Universal Robots URScript: Main Program Right.script

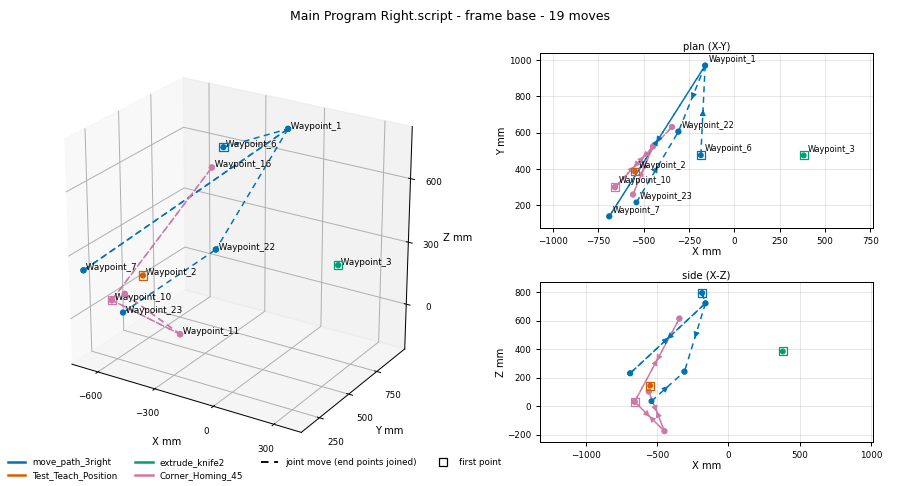
[picture p0: tool path of Main Program Right.script in frame base, 19 of 66 moves have a stored position in this frame; points joined in program order, loops and branches not executed]
def Main_Program_Right():
  global _hidden_verificationVariable=0
  set_tcp(p[0.00157,-0.09008,0.25767,0.0,0.0,0.0])
  set_safety_mode_transition_hardness(1)
  set_tool_communication(False, 115200, 0, 1, 1.5, 3.5)
  set_tool_output_mode(0)
  set_tool_digital_output_mode(0, 1)
  set_tool_digital_output_mode(1, 1)
  set_tool_voltage(0)
  set_target_payload(8.250000, [-0.001000, -0.057000, 0.067000], [0.051851, 0.051851, 0.051851, 0.000000, 0.000000, 0.000000])
  set_standard_analog_input_domain(0, 1)
  set_standard_analog_input_domain(1, 1)
  set_tool_analog_input_domain(0, 1)
  set_tool_analog_input_domain(1, 1)
  set_analog_outputdomain(0, 0)
  set_analog_outputdomain(1, 0)
  set_input_actions_to_default()
  set_gravity([0.0, 0.0, 9.82])
  global Point_1=p[0.0,0.0,0.0,0.0,0.0,0.0]
  # begin: URCap Installation Node
  #   Source: MachineLogic for Universal Robots, 3.1.7, Vention Inc.
  #   Type: MachineLogic for Universal Robots
  def waitForResponse(expected_response_vention, cname_vention):
  response_vention = socket_read_string(cname_vention,timeout=15)
  while response_vention != expected_response_vention:
  sleep(0.01)
  response_vention = socket_read_string(cname_vention,timeout=15)
  end
  sleep(0.01)
  sync()
  end
  def sendString(string_vention, expected_response_vention, cname_vention):
  socket_send_string(str_cat(string_vention,";"), cname_vention)
  response_vention = socket_read_string(cname_vention,timeout=15)
  if(response_vention == "nAck"):
  popup("nAck received")
  end
  while response_vention != expected_response_vention:
  sleep(0.01)
  response_vention = socket_read_string(cname_vention,timeout=15)
  if(response_vention == "nAck"):
  popup("nAck received")
  end
  end
  sleep(0.01)
  sync()
  end
  def sendStringNAck(string_vention, expected_response_vention, cname_vention):
  socket_send_string(str_cat(string_vention,";"), cname_vention)
  response_vention = socket_read_string(cname_vention,timeout=15)
  if(response_vention == "nAck"):
  popup("nAck received")
  end
  while(response_vention != expected_response_vention and response_vention != "nAck"):
  sleep(0.01)
  response_vention = socket_read_string(cname_vention,timeout=15)
  if(response_vention == "nAck"):
  popup("nAck received",blocking=True)
  end
  end
  sleep(0.01)
  sync()
  end
  def sendStringWithTimeout(string_vention, expected_response_vention, cname_vention):
  socket_send_string(str_cat(string_vention,";"), cname_vention)
  response_vention = socket_read_string(cname_vention,timeout=10)
  if(response_vention == "nAck"):
  popup("nAck received"+string_vention)
  end
  sleep(0.01)
  sync()
  end
  def pollString(string_vention, expected_response_vention, cname_vention):
  socket_send_string(str_cat(string_vention,";"), cname_vention)
  response_vention = socket_read_string(cname_vention,timeout=15)
  if(response_vention == "nAck"):
  popup("nAck received")
  end
  while response_vention != expected_response_vention:
  sleep(1)
  socket_send_string(str_cat(string_vention,";"), cname_vention)
  response_vention = socket_read_string(cname_vention,timeout=15)
  if(response_vention == "nAck"):
  popup("nAck received")
  end
  end
  sleep(0.01)
  sync()
  end
  def sendVariable(var_vention, data_vention, expected_response_vention, cname_vention):
  socket_set_var(var_vention, data_vention, cname_vention)
  response_vention = socket_read_string(cname_vention,timeout=15)
  if(response_vention == "nAck"):
  popup("nAck received")
  end
  while response_vention != expected_response_vention:
  sleep(0.01)
  response_vention = socket_read_string(cname_vention,timeout=15)
  if(response_vention == "nAck"):
  popup("nAck received")
  end
  end
  sleep(0.01)
  sync()
  end
  def intToString(integer_vention,cname_vention):
  stringFix=""
  multiplier_vention123=1
  if integer_vention<0:
  stringFix="-"
  multiplier_vention123=-1
  end
  socket_set_var("GetString",integer_vention*multiplier_vention123,cname_vention)
  string_vention=""
  while string_vention=="":
  sleep(0.01)
  string_vention=socket_read_string(cname_vention,timeout=15)
  end
  sleep(0.01)
  sync()
  string_vention=stringFix+string_vention
  return string_vention
  end
  string_vention=""
  isVentionMovementBusy = False
  isVentionParallelMovementSendingScript = False
  ventionThreadHandle = 1
  isVentionMovementBusyMachineMotion1 = False
  isVentionParallelMovementSendingScriptMachineMotion1 = False
  socket_vention = socket_open("192.168.3.52", 9999, "MachineMotion1")
  if socket_vention==False:
  popup("Check configuration, can't connect to MachineMotion")
  end
  waitForResponse("MachineMotion connection established", "MachineMotion1")
  sendString("isReady", "MachineMotion isReady = true", "MachineMotion1")
  sendStringWithTimeout("setURCapVersion2", "setURCapVersion loaded", "MachineMotion1")
  sendString("SET speed_v2 1000000", "Ack", "MachineMotion1")
  sendString("SET acceleration_v2 100000", "Ack", "MachineMotion1")
  sendString("SET de_axis_1_microsteps_config 8", "Ack", "MachineMotion1")
  sendString("SET de_axis_1_mechanical_gain_config_v2 150000.0", "Ack", "MachineMotion1")
  sendString("SET de_axis_1_direction_config 1", "Ack", "MachineMotion1")
  sendString("SET de_axis_1_type_config Custom Actuator ", "Ack", "MachineMotion1")
  sendString("de_axis_1_config_exec", "Ack", "MachineMotion1")
  # end: URCap Installation Node
  # begin: URCap Installation Node
  #   Source: WireTank Serial, 4.8.0, WireTank, LLC
  #   Type: WireTank Serial
  WTSerialBridge = rpc_factory("xmlrpc","http://127.0.0.1:40511/RPC2")
  # end: URCap Installation Node
  step_count_51af8de3_71b6_4904_b866_4a648f97dfbd = 0.0
  thread Step_Counter_Thread_b894e04d_ed7b_4f14_91e2_7b90849917c2():
    while (True):
      step_count_51af8de3_71b6_4904_b866_4a648f97dfbd = step_count_51af8de3_71b6_4904_b866_4a648f97dfbd + 1.0
      sync()
    end
  end
  run Step_Counter_Thread_b894e04d_ed7b_4f14_91e2_7b90849917c2()
  global freedrive_m_var=  False
  global thread2trigger=  False
  global Waypoint_6_p=p[-.184857361379, .475907634298, .794864406022, -.224954183187, -1.929458896935, .684866995731]
  global Waypoint_6_q=[-2.3977788130389612, -1.5333859895220776, 2.098509136830465, 0.9648317533680419, -0.8855178991900843, -0.44068843523134404]
  global Waypoint_1_p=p[-.161036555831, .970524399959, .722042384791, -.554954311189, .106465018540, .328580879483]
  global Waypoint_1_q=[-1.3071630636798304, -1.3366777312806626, 2.2083633581744593, 3.7187773424335937, -2.9519384543048304, 0.9132363796234131]
  global Waypoint_7_p=p[-.689650873132, .138963273545, .230691387978, -.851994598965, -1.645998530536, 1.646007616333]
  global Waypoint_7_q=[-0.9414032141314905, -1.501500443821289, 2.801856819783346, 4.981602895050802, -4.698942009602682, 1.571649193763733]
  global Waypoint_8_p=p[-.689650873132, .138963273545, .230691387978, -.851994598965, -1.645998530536, 1.646007616333]
  global Waypoint_8_q=[-0.9414032141314905, -1.501500443821289, 2.801856819783346, 4.981602895050802, -4.698942009602682, 1.571649193763733]
  global Waypoint_9_p=p[-.161036555831, .970524399959, .722042384791, -.554954311189, .106465018540, .328580879483]
  global Waypoint_9_q=[-1.3071630636798304, -1.3366777312806626, 2.2083633581744593, 3.7187773424335937, -2.9519384543048304, 0.9132363796234131]
  global Waypoint_22_p=p[-.308534453517, .606084664264, .242393158856, 1.369873371142, 1.066881263643, -1.257197506198]
  global Waypoint_22_q=[-1.4685500303851526, -0.9664557737163086, 1.6195090452777308, 0.9282776552387695, 1.6574476957321167, 0.2630845010280609]
  global Waypoint_23_p=p[-.540166575654, .215949141041, .034631452617, -1.505795438113, 1.057579835594, 1.573514753692]
  global Waypoint_23_q=[-0.46167117754091436, -1.1365486842444916, 2.508885685597555, 0.15223841249432368, 1.4952874183654785, 3.819530963897705]
  global Waypoint_24_p=p[-.308525559537, .606096497354, .242373144855, -2.133742737559, .349425192770, 2.130939839044]
  global Waypoint_24_q=[-1.8709262053119105, -1.2877716285041352, 2.192875687276022, 0.7510036665150146, 1.5878156423568726, 1.5091480016708374]
  global Waypoint_2_p=p[-.548957282596, .386284559177, .143710178207, 1.570800598292, -.000025190822, .000004803470]
  global Waypoint_2_q=[-1.0516188780414026, -1.010990933781006, 2.1562450567828577, -1.143702046280243, -1.0526168982135218, -0.0017235914813440445]
  global Waypoint_3_p=p[.382320178964, .475080148289, .384014983870, 1.881213850562, 2.483463485094, .075780854208]
  global Waypoint_3_q=[-3.0947259108172815, -1.8717390499510707, 2.1334107557879847, -0.21609540403399663, -0.2287352720843714, -0.09839088121523076]
  def calculate_point_to_move_towards(feature, direction, position_distance):
    local posDir=[direction[0], direction[1], direction[2]]
    if (norm(posDir) < 1e-6):
      return get_target_waypoint()
    end
    local direction_vector_normalized=normalize(posDir)
    local displacement_pose=p[direction_vector_normalized[0] * position_distance,direction_vector_normalized[1] * position_distance,direction_vector_normalized[2] * position_distance,0,0,0]
    local wanted_displacement_in_base_frame=pose_sub(pose_trans(feature, displacement_pose), feature)
    return pose_add(get_target_waypoint(), wanted_displacement_in_base_frame)
  end
  global Waypoint_10_p=p[-.658264763546, .299530128456, .030909835036, .426821001551, -1.621505068649, .437070885767]
  global Waypoint_10_q=[-1.350241486226217, -0.9702387017062684, 2.492185179387228, -1.7834822140135707, -0.33723670641054326, 1.8489984273910522]
  global Waypoint_11_p=p[-.448862677341, .524599667441, -.175967040878, 2.473330473302, -1.874382924863, .205319206046]
  global Waypoint_11_q=[-1.1354392210589808, -1.0039964479259034, 2.441021744404928, -2.875528474847311, -1.6043828169452112, 1.7329596281051636]
  global Waypoint_12_p=p[-.559130451394, .259233925829, .102445980692, -.822649281727, -1.486064670292, -.881476138414]
  global Waypoint_12_q=[-0.556256119404928, -1.0744255942157288, 2.9114087263690394, -1.7763501606383265, -4.185837809239523, 1.5288889408111572]
  global Waypoint_13_p=p[-.559130451394, .259233925829, .102445980692, -.822649281727, -1.486064670292, -.881476138414]
  global Waypoint_13_q=[-0.556256119404928, -1.0744255942157288, 2.9114087263690394, -1.7763501606383265, -4.185837809239523, 1.5288889408111572]
  global Waypoint_14_p=p[-.448862677341, .524599667441, -.175967040878, 2.473330473302, -1.874382924863, .205319206046]
  global Waypoint_14_q=[-1.1354392210589808, -1.0039964479259034, 2.441021744404928, -2.875528474847311, -1.6043828169452112, 1.7329596281051636]
  global Waypoint_15_p=p[-.658264763546, .299530128456, .030909835036, .426821001551, -1.621505068649, .437070885767]
  global Waypoint_15_q=[-1.350241486226217, -0.9702387017062684, 2.492185179387228, -1.7834822140135707, -0.33723670641054326, 1.8489984273910522]
  global Waypoint_16_p=p[-.343952006273, .632142227752, .615174722549, -.025948978133, -.008794819136, -.567469912202]
  global Waypoint_16_q=[-1.350241486226217, -0.9702451390079041, 2.492171827946798, -3.0669099293150843, 1.575993537902832, 2.355180025100708]
  global Waypoint_17_p=p[-.343952006273, .632142227752, .615174722549, -.025948978133, -.008794819136, -.567469912202]
  global Waypoint_17_q=[-1.350241486226217, -0.9702451390079041, 2.492171827946798, -3.0669099293150843, 1.575993537902832, 2.355180025100708]
  global Waypoint_18_p=p[-.658264763546, .299530128456, .030909835036, .426821001551, -1.621505068649, .437070885767]
  global Waypoint_18_q=[-1.350241486226217, -0.9702387017062684, 2.492185179387228, -1.7834822140135707, -0.33723670641054326, 1.8489984273910522]
  def move_path_3right():
    $ 20 "move_path_3right" "noBreak"
    $ 21 "'this is the path for Down, Over, then Back Around'"
    # 'this is the path for Down, Over, then Back Around'
    $ 22 "Comment"
    # Comment
    $ 23 "Home"
    movej([-3.4579734502641006, -2.05691362454537, 2.326567589830591, -0.22707360390354125, -0.19934432301767302, -0.10534790278823536], a=1.3962634015954636, v=1.0471975511965976)
    $ 24 "MoveJ"
    $ 25 "Waypoint_6" "breakAfter"
    movej(get_inverse_kin(Waypoint_6_p, qnear=Waypoint_6_q), a=1.3962634015954636, v=1.0471975511965976)
    $ 26 "Waypoint_1" "breakAfter"
    movej(get_inverse_kin(Waypoint_1_p, qnear=Waypoint_1_q), a=1.3962634015954636, v=1.0471975511965976)
    $ 27 "Waypoint_7" "breakAfter"
    movej(get_inverse_kin(Waypoint_7_p, qnear=Waypoint_7_q), a=1.3962634015954636, v=1.0471975511965976)
    $ 32 "Comment"
    # Comment
    $ 33 "p1≔pathturn[0]"
    global p1=pathturn[0]
    $ 34 "p2≔pathturn[1]"
    global p2=pathturn[1]
    $ 35 "p4≔pathturn[2]"
    global p4=pathturn[2]
    $ 36 "p5≔pathturn[3]"
    global p5=pathturn[3]
    $ 37 "MoveJ"
    $ 38 "p1" "breakAfter"
    movej(p1, a=1.3962634015954636, v=1.0471975511965976)
    $ 39 "Wait: 8.0"
    sleep(8.0)
    # begin: URCap Program Node
    #   Source: WireTank Serial, 4.8.0, WireTank, LLC
    #   Type: WireTank Serial
    $ 40 "Serial Bridge uR1"
    SerialResponse = WTSerialBridge.send_command("/dev/ttyUSB0",1200, 8, "None", "One", "None", 5000, "None", "None", [252,82,49], False)
    # end: URCap Program Node
    $ 41 "Wait: 1.0"
    sleep(1.0)
    $ 42 "MoveL"
    $ 43 "p2" "breakAfter"
    movel(p2, a=0.1, v=0.01)
    # begin: URCap Program Node
    #   Source: WireTank Serial, 4.8.0, WireTank, LLC
    #   Type: WireTank Serial
    $ 44 "Serial Bridge uR0"
    SerialResponse = WTSerialBridge.send_command("/dev/ttyUSB0",1200, 8, "None", "One", "None", 5000, "None", "None", [252,82,48], False)
    # end: URCap Program Node
    $ 45 "Wait: 0.5"
    sleep(0.5)
    $ 47 "MoveL"
    $ 48 "p4" "breakAfter"
    movel(p4, a=0.01, v=0.12)
    # begin: URCap Program Node
    #   Source: WireTank Serial, 4.8.0, WireTank, LLC
    #   Type: WireTank Serial
    $ 49 "Serial Bridge uR1"
    SerialResponse = WTSerialBridge.send_command("/dev/ttyUSB0",1200, 8, "None", "One", "None", 5000, "None", "None", [252,82,49], False)
    # end: URCap Program Node
    $ 50 "Wait: 1.0"
    sleep(1.0)
    $ 51 "MoveL"
    $ 52 "p5" "breakAfter"
    movel(p5, a=0.1, v=0.01)
    # begin: URCap Program Node
    #   Source: WireTank Serial, 4.8.0, WireTank, LLC
    #   Type: WireTank Serial
    $ 53 "Serial Bridge uR0"
    SerialResponse = WTSerialBridge.send_command("/dev/ttyUSB0",1200, 8, "None", "One", "None", 5000, "None", "None", [252,82,48], False)
    # end: URCap Program Node
    $ 54 "Wait: 2.0"
    sleep(2.0)
    $ 55 "Comment"
    # Comment
    $ 56 "pret1≔p[p5[0]+.1,p5[1],p5[2],p5[3],p5[4],p5[5]]"
    global pret1=p[p5[0]+.1,p5[1],p5[2],p5[3],p5[4],p5[5]]
    $ 57 "p_1≔pathturn[4]"
    global p_1=pathturn[4]
    $ 58 "p_2≔pathturn[5]"
    global p_2=pathturn[5]
    $ 59 "p_3≔pathturn[6]"
    global p_3=pathturn[6]
    $ 60 "p_4≔pathturn[7]"
    global p_4=pathturn[7]
    $ 61 "p_5≔pathturn[8]"
    global p_5=pathturn[8]
    $ 62 "p_preheat≔p[p_3[0]+.01,p_3[1],p_3[2],p_3[3],p_3[4],p_3[5]]"
    global p_preheat=p[p_3[0]+.01,p_3[1],p_3[2],p_3[3],p_3[4],p_3[5]]
    $ 63 "p_pre_ret≔p[p_3[0]+.1,p_3[1]+.1,p_3[2],p_2[3],p_2[4],p_2[5]]"
    global p_pre_ret=p[p_3[0]+.1,p_3[1]+.1,p_3[2],p_2[3],p_2[4],p_2[5]]
    $ 64 "p_pre_ret2≔p[p_3[0]+.1,p_3[1],p_3[2],p_3[3],p_3[4],p_3[5]]"
    global p_pre_ret2=p[p_3[0]+.1,p_3[1],p_3[2],p_3[3],p_3[4],p_3[5]]
    $ 65 "MoveJ"
    $ 66 "pret1" "breakAfter"
    movej(pret1, a=1.3962634015954636, v=1.3962634015954636)
    $ 67 "Waypoint_8" "breakAfter"
    movej(get_inverse_kin(Waypoint_8_p, qnear=Waypoint_8_q), a=1.3962634015954636, v=1.0471975511965976)
    $ 68 "Waypoint_9" "breakAfter"
    movej(get_inverse_kin(Waypoint_9_p, qnear=Waypoint_9_q), a=1.3962634015954636, v=1.3962634015954636)
    $ 69 "Waypoint_22" "breakAfter"
    movej(get_inverse_kin(Waypoint_22_p, qnear=Waypoint_22_q), a=1.3962634015954636, v=1.3962634015954636)
    $ 70 "'preheat'"
    # 'preheat'
    $ 71 "MoveJ"
    $ 72 "p_pre_ret" "breakAfter"
    movej(p_pre_ret, a=1.3962634015954636, v=1.0471975511965976)
    $ 73 "p_pre_ret2" "breakAfter"
    movej(p_pre_ret2, a=1.3962634015954636, v=1.0471975511965976)
    $ 74 "p_preheat" "breakAfter"
    movej(p_preheat, a=1.3962634015954636, v=1.0471975511965976)
    $ 75 "Wait: 8.0"
    sleep(8.0)
    $ 76 "MoveJ"
    $ 77 "p_pre_ret2" "breakAfter"
    movej(p_pre_ret2, a=1.3962634015954636, v=1.0471975511965976)
    $ 78 "p_pre_ret" "breakAfter"
    movej(p_pre_ret, a=1.3962634015954636, v=1.0471975511965976)
    $ 79 "Set"
    set_tcp(p[0.00662,-0.33062,0.10207,1.2092,-1.2092,1.2092])
    $ 80 "MoveL"
    $ 81 "p_1" "breakAfter"
    movel(p_1, a=1.2, v=0.05)
    # begin: URCap Program Node
    #   Source: WireTank Serial, 4.8.0, WireTank, LLC
    #   Type: WireTank Serial
    $ 82 "Serial Bridge uR1"
    SerialResponse = WTSerialBridge.send_command("/dev/ttyUSB0",1200, 8, "None", "One", "None", 5000, "None", "None", [252,82,49], False)
    # end: URCap Program Node
    $ 83 "Wait: 1.0"
    sleep(1.0)
    $ 84 "MoveL"
    $ 85 "p_2" "breakAfter"
    movel(p_2, a=1.2, v=0.01)
    $ 86 "MoveP"
    $ 87 "CircleMove"
    $ 88 "p_3" "noBreak"
    $ 89 "p_4" "breakAfter"
    movec(p_3, p_4, a=0.01, v=5.0E-4, r=0.0, mode=1)
    $ 90 "MoveL"
    $ 91 "p_5" "breakAfter"
    movel(p_5, a=1.2, v=0.012)
    # begin: URCap Program Node
    #   Source: WireTank Serial, 4.8.0, WireTank, LLC
    #   Type: WireTank Serial
    $ 92 "Serial Bridge uR0"
    SerialResponse = WTSerialBridge.send_command("/dev/ttyUSB0",1200, 8, "None", "One", "None", 5000, "None", "None", [252,82,48], False)
    # end: URCap Program Node
    $ 93 "Wait: 2.0"
    sleep(2.0)
    $ 94 "MoveL"
    $ 95 "Waypoint_23" "breakAfter"
    movel(Waypoint_23_p, a=1.2, v=0.25)
    $ 96 "MoveJ"
    $ 97 "Waypoint_24" "breakAfter"
    movej(get_inverse_kin(Waypoint_24_p, qnear=Waypoint_24_q), a=1.3962634015954636, v=1.0471975511965976)
    $ 98 "Comment"
    # Comment
    $ 99 "Comment"
    # Comment
    $ 100 "Comment"
    # Comment
    $ 101 "Comment"
    # Comment
    $ 102 "Comment"
    # Comment
    $ 103 "Comment"
    # Comment
    $ 104 "Comment"
    # Comment
    $ 105 "Home"
    movej([-3.4579734502641006, -2.05691362454537, 2.326567589830591, -0.22707360390354125, -0.19934432301767302, -0.10534790278823536], a=1.3962634015954636, v=1.0471975511965976)
  end
  def Test_Teach_Position():
    $ 106 "Test_Teach_Position" "noBreak"
    $ 107 "Home"
    movej([-3.4579734502641006, -2.05691362454537, 2.326567589830591, -0.22707360390354125, -0.19934432301767302, -0.10534790278823536], a=1.3962634015954636, v=1.0471975511965976)
    $ 111 "MoveJ"
    $ 112 "Waypoint_2" "breakAfter"
    set_tcp(p[0.0,0.0,0.019,0.0,0.0,0.0])
    movej(get_inverse_kin(Waypoint_2_p, qnear=Waypoint_2_q), a=1.3962634015954636, v=1.0471975511965976)
    $ 113 "freedrive_m_var≔ False "
    global freedrive_m_var=  False
    $ 114 "freedrive_m_var≔ True "
    global freedrive_m_var=  True
    $ 115 "Popup: Move the robot to the peg center, then click 'Continue'"
    popup("Move the robot to the peg center, then click 'Continue'", "Message", False, False, blocking=True)
    $ 116 "freedrive_m_var≔ False "
    global freedrive_m_var=  False
    $ 117 "Wait: 0.25"
    sleep(0.25)
    $ 118 "sync()"
    sync()
    $ 119 "tcp_pose≔get_actual_joint_positions()"
    global tcp_pose= get_actual_joint_positions ()
  end
  def align_tcp_left():
    $ 162 "align_tcp_left" "noBreak"
    $ 163 "'this program aligns the tcp parallel to the y direction'"
    # 'this program aligns the tcp parallel to the y direction'
    $ 164 "cp≔get_actual_tcp_pose()"
    global cp= get_actual_tcp_pose ()
    $ 165 "aligned_y_pose≔p[cp[0],cp[1],cp[2],1.570796,0,0]"
    global aligned_y_pose=p[cp[0],cp[1],cp[2],1.570796,0,0]
    $ 166 "MoveJ"
    $ 167 "aligned_y_pose" "breakAfter"
    movej(aligned_y_pose, a=1.3962634015954636, v=1.0471975511965976)
  end
  def extrude_knife2():
    $ 168 "extrude_knife2" "noBreak"
    $ 169 "Home"
    movej([-3.4579734502641006, -2.05691362454537, 2.326567589830591, -0.22707360390354125, -0.19934432301767302, -0.10534790278823536], a=1.3962634015954636, v=1.0471975511965976)
    $ 170 "Set"
    set_tcp(p[-0.00438,-0.33062,0.10207,1.2092,-1.2092,1.2092])
    $ 171 "MoveJ"
    $ 172 "Waypoint_3" "breakAfter"
    movej(get_inverse_kin(Waypoint_3_p, qnear=Waypoint_3_q), a=1.3962634015954636, v=1.0471975511965976)
    $ 173 "'extrude out a foot'"
    # 'extrude out a foot'
    # begin: URCap Program Node
    #   Source: WireTank Serial, 4.8.0, WireTank, LLC
    #   Type: WireTank Serial
    $ 174 "Serial Bridge uR1"
    SerialResponse = WTSerialBridge.send_command("/dev/ttyUSB0",1200, 8, "None", "One", "None", 5000, "None", "None", [252,82,49], False)
    # end: URCap Program Node
    $ 175 "Wait: 24.0"
    sleep(24.0)
    # begin: URCap Program Node
    #   Source: WireTank Serial, 4.8.0, WireTank, LLC
    #   Type: WireTank Serial
    $ 176 "Serial Bridge uR0"
    SerialResponse = WTSerialBridge.send_command("/dev/ttyUSB0",1200, 8, "None", "One", "None", 5000, "None", "None", [252,82,48], False)
    # end: URCap Program Node
    $ 177 "Popup: grab extrusion then press ok"
    popup("grab extrusion then press ok", "Message", False, False, blocking=True)
    $ 178 "Home"
    movej([-3.4579734502641006, -2.05691362454537, 2.326567589830591, -0.22707360390354125, -0.19934432301767302, -0.10534790278823536], a=1.3962634015954636, v=1.0471975511965976)
  end
  def align_tcp_forward():
    $ 179 "align_tcp_forward" "noBreak"
    $ 180 "'this program aligns the tcp parallel to the y direction'"
    # 'this program aligns the tcp parallel to the y direction'
    $ 181 "cp≔get_actual_tcp_pose()"
    global cp= get_actual_tcp_pose ()
    $ 182 "aligned_y_pose≔p[cp[0],cp[1],cp[2],0,-1.570796,0]"
    global aligned_y_pose=p[cp[0],cp[1],cp[2],0,-1.570796,0]
    $ 183 "MoveJ"
    $ 184 "aligned_y_pose" "breakAfter"
    movej(aligned_y_pose, a=1.3962634015954636, v=1.0471975511965976)
  end
  def align_tcp_up():
    $ 185 "align_tcp_up" "noBreak"
    $ 186 "'this program aligns the tcp parallel to the y direction'"
    # 'this program aligns the tcp parallel to the y direction'
    $ 187 "cp≔get_actual_tcp_pose()"
    global cp= get_actual_tcp_pose ()
    $ 188 "aligned_y_pose≔p[cp[0],cp[1],cp[2],0,0,0]"
    global aligned_y_pose=p[cp[0],cp[1],cp[2],0,0,0]
    $ 189 "MoveJ"
    $ 190 "aligned_y_pose" "breakAfter"
    movej(aligned_y_pose, a=1.3962634015954636, v=1.0471975511965976)
  end
  def Corner_Homing_45():
    $ 191 "Corner_Homing_45" "noBreak"
    $ 192 "'Use this program when tool is already positioned close to corner at 45deg'"
    # 'Use this program when tool is already positioned close to corner at 45deg'
    $ 193 "'tool flange will seek all 3 sides. will save those 5 locs in p__'"
    # 'tool flange will seek all 3 sides. will save those 5 locs in p__'
    $ 194 "Set"
    set_tcp(p[0.00157,-0.09008,0.25767,0.0,0.0,0.0])
    $ 195 "'dummy move below for debug'"
    # 'dummy move below for debug'
    $ 200 "Wait: 1.0"
    sleep(1.0)
    $ 201 "tp≔get_actual_tcp_pose()"
    global tp= get_actual_tcp_pose ()
    $ 202 "Script: analyze_touchpoints.script"
    # this file creates the function for analyzing touchpoints
    # define pi
    pi = 3.1415926535

    # this is the main entry point for calculations.
    # it takes in the 5 points, analyzes the shape of the box, and then calculates path points and returns them
    # specifically for Down, Over, then Around (DOtA)
    # specifically for right-sided boxes (vertical weld on right side of edge)
    def main_calculate_right(p11, p12, p21, p22, p3):
        struct1 = analyze_touchpoints_only(p11, p12, p21, p22, p3)
        struct2 = calculate_DOtA_points_right(struct1)
        return struct2
    end

    # this is the main entry point for calculations.
    # it takes in the 5 points, analyzes the shape of the box, and then calculates path points and returns them
    # specifically for Down, Over, then Around (DOtA)
    # specifically for left-sided boxes (vertical weld on left side of edge)
    def main_calculate_left(p11, p12, p21, p22, p3):
        struct1 = analyze_touchpoints_only(p11, p12, p21, p22, p3)
        struct2 = calculate_DOtA_points_left(struct1)
        return struct2
    end

    # it takes 5 arguments as points
    # it returns a struct containing: (pointintersect, pointapproach1, pointapproach2, point1, point2, point3, point4, point5, pointreturn1, heading1, heading2, heading3, path2r1, path2r2, path2l1, path2l2)
    # specifically for Around then Up (AtU)
    def analyze_touchpoints(p11, p12, p21, p22, p3):
      # FIND THE INTERSECTION
      # comment get the z
      zcoord=p3[2]

      # get the raw points from the first line
      l1p1x=p11[0]
      l1p1y=p11[1]
      l1p2x=p12[0]
      l1p2y=p12[1]

      # equate the first line in 2d space
      ml1 = (l1p2y-l1p1y) / (l1p2x-l1p1x)

      # b = y - mx
      bl1 = l1p1y - ml1 * l1p1x

      # get the raw points from the second line
      l2p1x=p21[0]
      l2p1y=p21[1]
      l2p2x=p22[0]
      l2p2y=p22[1]

      # equate the second line in 2d space
      ml2 = (l2p2y-l2p1y) / (l2p2x-l2p1x)

      # b = y - mx
      bl2 = l2p1y - ml2 * l2p1x


      # find the intersection of the two lines
      # m1x+b1 = m2x+b2
      # m1x - m2x = b2 - b1
      # x = (b2-b1) / (m1-m2)
      xintersect = (bl2-bl1) / (ml1-ml2)
      yintersect = ml1 * xintersect + bl1

      #FIND THE VECTORS
      #define a vector from the intersection to the second point on the first line
      l1delxfull = l1p2x - xintersect
      l1delyfull = l1p2y - yintersect

      l1delmag = sqrt(l1delxfull*l1delxfull + l1delyfull*l1delyfull)

      l1delxunit = l1delxfull / l1delmag
      l1delyunit = l1delyfull / l1delmag

      #define a vector from the intersection to the second point on the second line
      l2delxfull = l2p2x - xintersect
      l2delyfull = l2p2y - yintersect

      l2delmag = sqrt(l2delxfull*l2delxfull + l2delyfull*l2delyfull)

      l2delxunit = l2delxfull / l2delmag
      l2delyunit = l2delyfull / l2delmag

      # FIND THE FOUR POINTS ON THE LINES
      # find locations 8 inches away from  intersect point
      # CONST
      welddistance = 8
      roundoverdistance = 0.05
      zup = .375
      # inches
      wd = welddistance * 25.4 / 1000
      rod = roundoverdistance * 25.4 / 1000
      zup = zup * 25.4 / 1000

      # now we have the unit vector. extend the weld distance from the intersection
      x = xintersect + l1delxunit * wd
      y = yintersect + l1delyunit * wd
      z = zcoord + zup

      point1 = p[x,y,z,1.570796,0,0] # dummy orientation for now

      x = xintersect + l1delxunit * rod
      y = yintersect + l1delyunit * rod

      point2 = p[x,y,z,1.570796,0,0]

      # now we have the unit vector. extend the weld distance from the intersection
      x = xintersect + l2delxunit * wd
      y = yintersect + l2delyunit * wd

      point5 = p[x,y,z,0,-1.570796,0]

      x = xintersect + l2delxunit * rod
      y = yintersect + l2delyunit * rod

      point4 = p[x,y,z,0,-1.570796,0]

      #DEFINE APPROACH POINTS
      pointintersect = p[xintersect,yintersect,zcoord,0,0,0]
      pointapproach1 = p[xintersect+0.1,yintersect+0.1,z,1.570796,0,0]
      pointapproach2 = p[point1[0], point1[1]+0.1, point1[2], point1[3], point1[4], point1[5]]
      pointreturn1 = p[point5[0]+0.1, point5[1], point5[2], point5[3], point5[4], point5[5]]

      #FIND HEADINGS
      #for each heading, find the angle of the line with respect to the pos x axis. then add/subtract 90 degrees because you want to be perpendicular to that
      headingvector1 = convert_uv_to_heading(l1delxunit, l1delyunit)
      headingvector2 = convert_uv_to_heading(l2delxunit, l2delyunit)
      # find halfway heading
      heading2 = (headingvector1 + headingvector2)/2
      # find headings that the robot should face while traveling, perpendicular to the vectors of the sides of the box
      heading1 = headingvector1 + pi/2
      heading3 = headingvector2 - pi/2

      #FIND POINT 3
      #see if we have to / can find point 3
      findpoint3 = True
      if roundoverdistance == 0:
        findpoint3 = False
      end
      if findpoint3:
        # i need to find the point3 such that the arc from p2 to p3 to p4 is tangent to p1-p2 and p4-p5. making this a smooth path will be good
        # the direction of movement is from pointintersect in the direction of heading2
        # how much movement though? this will depend on whether it is actually a 90 degree angle or not.
        # first, find the perpendicular lines through points 2 and 4
        perp2 = find_perpendicular_line(ml1, point2[0], point2[1])
        perp4 = find_perpendicular_line(ml2, point4[0], point4[1])
        # next, find the intersection of those two lines
        perpintersect = find_intersection(perp2[0], perp2[1], perp4[0], perp4[1])
        radiusofcircle = distance_between(perpintersect[0], perpintersect[1], 0, point2[0], point2[1], 0)
        # find a vector the direction of heading2
        uvx = cos(heading2)
        uvy = sin(heading2)
        # compute point3. pass in negative radius because the direction is into the tank but we want to move from the intersection out to the rounded edge.
        point3coords = add_vectordistance_to_point(perpintersect[0], perpintersect[1], z, uvx, uvy, 0, -1 * radiusofcircle)
        point3 = p[point3coords[0], point3coords[1], point3coords[2], 0, 0, 0]
      end

      #APPLY ACTUAL RXRYRZ TO POINTS
      # convert the headings to rxryrz and insert those values into the relevant points
      rxryrz = convert_heading_to_axang(heading1)
      rx = rxryrz[0]
      ry = rxryrz[1]
      rz = rxryrz[2]
      pointapproach1 = p[pointapproach1[0], pointapproach1[1], pointapproach1[2], rx, ry, rz]
      pointapproach2 = p[pointapproach2[0], pointapproach2[1], pointapproach2[2], rx, ry, rz]
      point1 = p[point1[0], point1[1], point1[2], rx, ry, rz]
      point2 = p[point2[0], point2[1], point2[2], rx, ry, rz]
      rxryrz = convert_heading_to_axang(heading2)
      rx = rxryrz[0]
      ry = rxryrz[1]
      rz = rxryrz[2]
      if findpoint3:
        point3 = p[point3[0], point3[1], point3[2], rx, ry, rz]
      else:
        point3 = point2
      end
      rxryrz = convert_heading_to_axang(heading3)
      rx = rxryrz[0]
      ry = rxryrz[1]
      rz = rxryrz[2]
      point4 = p[point4[0], point4[1], point4[2], rx, ry, rz]
      point5 = p[point5[0], point5[1], point5[2], rx, ry, rz]
      pointreturn1 = p[pointreturn1[0], pointreturn1[1], pointreturn1[2], rx, ry, rz]

      #find path2 (the part that goes up)
      four_vertical_points = find_vertical_points(pointintersect, l1delxunit, l1delyunit, l2delxunit, l2delyunit, zup, wd, heading1, heading3)
      path2r1 = four_vertical_points[0]
      path2r2 = four_vertical_points[1]
      path2l1 = four_vertical_points[2]
      path2l2 = four_vertical_points[3]

      #RETURN STRUCT
      ret = struct(pointintersect=pointintersect, pointapproach1=pointapproach1, pointapproach2=pointapproach2, point1=point1, point2=point2, point3=point3, point4=point4, point5=point5, pointreturn1=pointreturn1, heading1=heading1, heading2=heading2, heading3=heading3, path2r1=path2r1, path2r2=path2r2, path2l1=path2l1, path2l2=path2l2)
      return ret
    end

    # it takes 5 arguments as points
    # it returns a struct containing: (pointintersect, heading1, heading2, heading3, l1delxunit, l1delyunit, l2delxunit, l2delyunit)
    def analyze_touchpoints_only(p11, p12, p21, p22, p3):
      # FIND THE INTERSECTION
      # comment get the z
      zcoord=p3[2]

      # get the raw points from the first line
      l1p1x=p11[0]
      l1p1y=p11[1]
      l1p2x=p12[0]
      l1p2y=p12[1]

      # equate the first line in 2d space
      ml1 = (l1p2y-l1p1y) / (l1p2x-l1p1x)

      # b = y - mx
      bl1 = l1p1y - ml1 * l1p1x

      # get the raw points from the second line
      l2p1x=p21[0]
      l2p1y=p21[1]
      l2p2x=p22[0]
      l2p2y=p22[1]

      # equate the second line in 2d space
      ml2 = (l2p2y-l2p1y) / (l2p2x-l2p1x)

      # b = y - mx
      bl2 = l2p1y - ml2 * l2p1x


      # find the intersection of the two lines
      # m1x+b1 = m2x+b2
      # m1x - m2x = b2 - b1
      # x = (b2-b1) / (m1-m2)
      xintersect = (bl2-bl1) / (ml1-ml2)
      yintersect = ml1 * xintersect + bl1

      pointintersect = p[xintersect,yintersect,zcoord,0,0,0]

      #FIND THE VECTORS
      #define a vector from the intersection to the second point on the first line
      l1delxfull = l1p2x - xintersect
      l1delyfull = l1p2y - yintersect

      l1delmag = sqrt(l1delxfull*l1delxfull + l1delyfull*l1delyfull)

      l1delxunit = l1delxfull / l1delmag
      l1delyunit = l1delyfull / l1delmag

      #define a vector from the intersection to the second point on the second line
      l2delxfull = l2p2x - xintersect
      l2delyfull = l2p2y - yintersect

      l2delmag = sqrt(l2delxfull*l2delxfull + l2delyfull*l2delyfull)

      l2delxunit = l2delxfull / l2delmag
      l2delyunit = l2delyfull / l2delmag

      #FIND HEADINGS
      #for each heading, find the angle of the line with respect to the pos x axis. then add/subtract 90 degrees because you want to be perpendicular to that
      headingvector1 = convert_uv_to_heading(l1delxunit, l1delyunit)
      headingvector2 = convert_uv_to_heading(l2delxunit, l2delyunit)
      # find halfway heading
      heading2 = (headingvector1 + headingvector2)/2
      # find headings that the robot should face while traveling, perpendicular to the vectors of the sides of the box
      heading1 = headingvector1 + pi/2
      heading3 = headingvector2 - pi/2

      #RETURN STRUCT
      ret = struct(pointintersect=pointintersect, heading1=heading1, heading2=heading2, heading3=heading3, l1delxunit=l1delxunit, l1delyunit=l1delyunit, l2delxunit=l2delxunit, l2delyunit=l2delyunit)
      return ret
    end

    # given a struct from analyze_touchpoints_only(), calculate the points
    def calculate_DOtA_points_right(struct1):
        # get the stuff from the struct
        pointintersect = struct1[0]
        heading1 = struct1[1]
        heading2 = struct1[2]
        heading3 = struct1[3]
        l1delxunit = struct1[4]
        l1delyunit = struct1[5]
        l2delxunit = struct1[6]
        l2delyunit = struct1[7]

        # FIND THE POINTS ON THE LINES OF THE FIRST TURN PATH
        # find locations 8 inches away from  intersect point
        # CONST
        welddistance1 = 8 # vertical weld distance
        welddistance2 = 3 # first path second leg
        welddistance3 = 8 # second path second leg
        zup = .375
        # inches
        wd1 = welddistance1 * 25.4 / 1000
        wd2 = welddistance2 * 25.4 / 1000
        wd3 = welddistance3 * 25.4 / 1000
        zup = zup * 25.4 / 1000

        x = pointintersect[0] + l1delxunit * zup
        y = pointintersect[1] + l1delyunit * zup
        z = pointintersect[2] + zup

        #apply actual rxryrz to points
        # convert the headings to rxryrz and insert those values into the relevant points
        rxryrz = convert_heading_to_axang_preheatdown(heading1)
        rx = rxryrz[0]
        ry = rxryrz[1]
        rz = rxryrz[2]

        point1 = p[x, y, z + wd1, rx, ry, rz]
        point2 = p[x, y, z, rx, ry, rz]

        # convert the headings to rxryrz and insert those values into the relevant points
        rxryrz = convert_heading_to_axang_ccw(heading1)
        rx = rxryrz[0]
        ry = rxryrz[1]
        rz = rxryrz[2]

        point4 = p[x, y, z, rx, ry, rz]
        x = x + l1delxunit * wd2
        y = y + l1delyunit * wd2
        point5 = p[x, y, z, rx, ry, rz]

        # FIND THE POINTS ON THE LINES OF THE SECOND AROUND PATH
        roundoverdistance = 0.05
        rod = roundoverdistance * 25.4 / 1000

        # now we have the unit vector. extend the weld distance from the intersection
        x = pointintersect[0] + l1delxunit * (zup)
        y = pointintersect[1] + l1delyunit * zup
        # convert the headings to rxryrz and insert those values into the relevant points
        rxryrz = convert_heading_to_axang(heading1)
        rx = rxryrz[0]
        ry = rxryrz[1]
        rz = rxryrz[2]
        point_1 = p[x, y, z, rx, ry, rz]

        x = pointintersect[0] + l1delxunit * rod
        y = pointintersect[1] + l1delyunit * rod
        point_2 = p[x, y, z, rx, ry, rz]

        # now we have the unit vector. extend the weld distance from the intersection
        x = pointintersect[0] + l2delxunit * wd3
        y = pointintersect[1] + l2delyunit * wd3
        # convert the headings to rxryrz and insert those values into the relevant points
        rxryrz = convert_heading_to_axang(heading3)
        rx = rxryrz[0]
        ry = rxryrz[1]
        rz = rxryrz[2]
        point_5 = p[x, y, z, rx, ry, rz]

        x = pointintersect[0] + l2delxunit * rod
        y = pointintersect[1] + l2delyunit * rod
        point_4 = p[x, y, z, rx, ry, rz]

        #FIND POINT 3
        # by calling analyze_touchpoints()
        atret = analyze_touchpoints(point_2, point_1, point_4, point_5, pointintersect)
        point_3 = atret[5]


        struct2 = struct(point1=point1, point2=point2, point4=point4, point5=point5, point_1=point_1, point_2=point_2, point_3=point_3, point_4=point_4, point_5=point_5)
        return struct2
    end

    # given a struct from analyze_touchpoints_only(), calculate the points
    def calculate_DOtA_points_left(struct1):
        # get the stuff from the struct
        pointintersect = struct1[0]
        heading1 = struct1[1]
        heading2 = struct1[2]
        heading3 = struct1[3]
        l1delxunit = struct1[4]
        l1delyunit = struct1[5]
        l2delxunit = struct1[6]
        l2delyunit = struct1[7]

        # FIND THE POINTS ON THE LINES OF THE FIRST TURN PATH
        # find locations 8 inches away from  intersect point
        # CONST
        welddistance = 8
        zup = .375
        # inches
        wd = welddistance * 25.4 / 1000
        zup = zup * 25.4 / 1000

        x = pointintersect[0] + l2delxunit * zup
        y = pointintersect[1] + l2delyunit * zup
        z = pointintersect[2] + zup

        #apply actual rxryrz to points
        # convert the headings to rxryrz and insert those values into the relevant points
        rxryrz = convert_heading_to_axang_preheatdown(heading3)
        rx = rxryrz[0]
        ry = rxryrz[1]
        rz = rxryrz[2]

        point1 = p[x, y, z + wd, rx, ry, rz]
        point2 = p[x, y, z, rx, ry, rz]

        # convert the headings to rxryrz and insert those values into the relevant points
        rxryrz = convert_heading_to_axang(heading3)
        rx = rxryrz[0]
        ry = rxryrz[1]
        rz = rxryrz[2]

        point4 = p[x, y, z, rx, ry, rz]
        x = x + l2delxunit * wd
        y = y + l2delyunit * wd
        point5 = p[x, y, z, rx, ry, rz]

        # FIND THE POINTS ON THE LINES OF THE SECOND AROUND PATH
        roundoverdistance = 0.05
        rod = roundoverdistance * 25.4 / 1000

        # now we have the unit vector. extend the weld distance from the intersection
        x = pointintersect[0] + l2delxunit * (zup)
        y = pointintersect[1] + l2delyunit * zup
        # convert the headings to rxryrz and insert those values into the relevant points
        rxryrz = convert_heading_to_axang_ccw(heading3)
        rx = rxryrz[0]
        ry = rxryrz[1]
        rz = rxryrz[2]
        point_1 = p[x, y, z, rx, ry, rz]

        x = pointintersect[0] + l2delxunit * rod
        y = pointintersect[1] + l2delyunit * rod
        point_2 = p[x, y, z, rx, ry, rz]

        # now we have the unit vector. extend the weld distance from the intersection
        x = pointintersect[0] + l1delxunit * wd
        y = pointintersect[1] + l1delyunit * wd
        # convert the headings to rxryrz and insert those values into the relevant points
        rxryrz = convert_heading_to_axang_ccw(heading1)
        rx = rxryrz[0]
        ry = rxryrz[1]
        rz = rxryrz[2]
        point_5 = p[x, y, z, rx, ry, rz]

        x = pointintersect[0] + l1delxunit * rod
        y = pointintersect[1] + l1delyunit * rod
        point_4 = p[x, y, z, rx, ry, rz]

        #FIND POINT 3
        # by calling analyze_touchpoints()
        atret = analyze_touchpoints(point_2, point_1, point_4, point_5, pointintersect)
        point_3 = atret[5]
        #point 3 will not have the correct rxryrz though because now the gun needs to be face up.
        rxryrz = convert_heading_to_axang_ccw(heading2)
        rx = rxryrz[0]
        ry = rxryrz[1]
        rz = rxryrz[2]
        point_3 = p[point_3[0], point_3[1], point_3[2], rx, ry, rz]

        struct2 = struct(point1=point1, point2=point2, point4=point4, point5=point5, point_1=point_1, point_2=point_2, point_3=point_3, point_4=point_4, point_5=point_5)
        return struct2
    end

    # given a heading, (ccw from +x axis), find the mx+b slope
    # fails if exactly vertical
    def get_slope_from_heading(heading):
        return tan(heading)
    end



    # this function finds the points (and rxryrz) of the 2 points (start and end) of vertical weld section
    def find_vertical_points(pointintersect, l1delxunit, l1delyunit, l2delxunit, l2delyunit, offset, wd, heading1, heading3):

      # find right side stuff
      # find the point in 3d space that is .375 up and .375 over
      x = pointintersect[0] + l1delxunit * offset
      y = pointintersect[1] + l1delyunit * offset
      z = pointintersect[2] + offset
      # find rxryrz
      rxryrz = convert_heading_to_axang_preheatup(heading1)
      rx = rxryrz[0]
      ry = rxryrz[1]
      rz = rxryrz[2]
      path2r1 = p[x, y, z, rx, ry, rz]
      path2r2 = p[x, y, z + wd, rx, ry, rz]

      # find left side
      # find the point in 3d space that is .375 up and .375 over
      x = pointintersect[0] + l2delxunit * offset
      y = pointintersect[1] + l2delyunit * offset
      z = pointintersect[2] + offset
      # find rxryrz
      rxryrz = convert_heading_to_axang_preheatup(heading3)
      rx = rxryrz[0]
      ry = rxryrz[1]
      rz = rxryrz[2]
      path2l1 = p[x, y, z, rx, ry, rz]
      path2l2 = p[x, y, z + wd, rx, ry, rz]

      ret = struct(path2r1=path2r1, path2r2=path2r2, path2l1=path2l1, path2l2=path2l2)
      return ret
    end

    # this function converts a unit vector to its heading angle ccw from x+ axis
    # takes uvx and uvy
    # returns heading in radians
    def convert_uv_to_heading(uvx, uvy):
      baseang = atan(uvy/uvx)
      if uvx < 0:
        ang = baseang + pi
      elif uvy < 0:
        ang = baseang + pi * 2
      else:
        ang = baseang
      end
      return ang
    end

    # this function finds the equation of a line, perpendicular to a given line, and going through a given point
    # takes 3 arguments: m (the original line's slope), x (point's x coord), y (point's y coord). the b of the original line is not needed
    # returns a list of [m,b] (the slope and intercept of the new line)
    def find_perpendicular_line(origm, x, y):
      m = (1/origm) * -1
      b = y - m*x
      ret = [m, b]
      return ret
    end

    # this function finds the intersection point between two lines in the xy plane
    # takes 4 arguments: m1, b1, m2, b2
    # returns a list of [x,y] (the point of intersection)
    def find_intersection(m1, b1, m2, b2):
      # m1x+b1 = m2x+b2
      # m1x - m2x = b2 - b1
      # x = (b2-b1) / (m1-m2)
      x = (b2-b1) / (m1-m2)
      y = m1 * x + b1
      ret = [x, y]
      return ret
    end

    # this function finds the distance between 2 points in 3d space
    # it takes 6 arguments: x1, y1, z1, x2, y2, z2
    # it returns a distance
    def distance_between(x1, y1, z1, x2, y2, z2):
      distsquared = (x2-x1)*(x2-x1)+(y2-y1)*(y2-y1)+(z2-z1)*(z2-z1)
      dist = sqrt(distsquared)
      return dist
    end

    # this function takes a point, a unit vector, and a distance, and adds the distance to the point in the direction of the unit vector (3d space)
    # it returns a point as a list of coordinates
    def add_vectordistance_to_point(xi, yi, zi, uvx, uvy, uvz, delta):
      xf = xi + uvx * delta
      yf = yi + uvy * delta
      zf = zi + uvz * delta
      ret = [xf, yf, zf]
      return ret
    end

    # this function converts a heading (ccw radians from the positive x axis) into rxryrz to be put into a point p[]
    # this will point the gun in this heading with the bottom side of the gun facing up.
    # the values used in this program were calculated by doing rotation matrix math in the file on WI-CALVINB10 C. Documents. Theory for converting rotations into axis angle representations
    def convert_heading_to_axang(heading):
     axisxraw = -1 * sin(heading)
     axisyraw = cos(heading) + 1
     axiszraw = sin(heading)

     magnitude = sqrt(axisxraw*axisxraw + axisyraw*axisyraw + axiszraw*axiszraw)

     axisxunit = axisxraw / magnitude
     axisyunit = axisyraw / magnitude
     axiszunit = axiszraw / magnitude

     angle = acos( (cos(heading) - 1) / 2 )

     rxout = axisxunit * angle
     ryout = axisyunit * angle
     rzout = axiszunit * angle

     return [rxout, ryout, rzout]
    end

    # this function converts a heading (ccw radians from the positive x axis) into rxryrz to be put into a point p[]
    # this will point the gun in this heading with the preheat side of the gun tip facing up. Used for welding in a vertical path.
    # the values used in this program were calculated by doing rotation matrix math in the file on WI-CALVINB10 C. Documents. Theory for converting rotations into axis angle representations
    def convert_heading_to_axang_preheatup(heading):
     axisxraw = -sin(heading) + 1
     axisyraw = cos(heading)
     axiszraw = cos(heading)

     magnitude = sqrt(axisxraw*axisxraw + axisyraw*axisyraw + axiszraw*axiszraw)

     axisxunit = axisxraw / magnitude
     axisyunit = axisyraw / magnitude
     axiszunit = axiszraw / magnitude

     angle = acos( (-sin(heading) - 1) / 2 )

     rxout = axisxunit * angle
     ryout = axisyunit * angle
     rzout = axiszunit * angle

     return [rxout, ryout, rzout]
    end

    # this function converts a heading (ccw radians from the positive x axis) into rxryrz to be put into a point p[]
    # this will point the gun in this heading with the preheat side of the gun tip facing down. Used for welding in a vertical path downwards.
    # the values used in this program were calculated by doing rotation matrix math in the file on WI-CALVINB10 C. Documents. Theory for converting rotations into axis angle representations
    def convert_heading_to_axang_preheatdown(heading):
     axisxraw = -sin(heading) - 1
     axisyraw = cos(heading)
     axiszraw = -cos(heading)

     magnitude = sqrt(axisxraw*axisxraw + axisyraw*axisyraw + axiszraw*axiszraw)

     axisxunit = axisxraw / magnitude
     axisyunit = axisyraw / magnitude
     axiszunit = axiszraw / magnitude

     angle = acos( (sin(heading) - 1) / 2 )

     rxout = axisxunit * angle
     ryout = axisyunit * angle
     rzout = axiszunit * angle

     return [rxout, ryout, rzout]
    end

    # this function converts a heading (ccw radians from the positive x axis) into rxryrz to be put into a point p[]
    # this will point the gun in this heading with the preheat side of the gun tip facing right. Used for welding counterclockwise around the box.
    # the values used in this program were calculated by doing rotation matrix math in the file on WI-CALVINB10 C. Documents. Theory for converting rotations into axis angle representations
    def convert_heading_to_axang_ccw(heading):
     axisxraw = -sin(heading)
     axisyraw = cos(heading) - 1
     axiszraw = -sin(heading)

     magnitude = sqrt(axisxraw*axisxraw + axisyraw*axisyraw + axiszraw*axiszraw)

     axisxunit = axisxraw / magnitude
     axisyunit = axisyraw / magnitude
     axiszunit = axiszraw / magnitude

     angle = acos( (-cos(heading) - 1) / 2 )

     rxout = axisxunit * angle
     ryout = axisyunit * angle
     rzout = axiszunit * angle

     return [rxout, ryout, rzout]
    end

    # this function is for getting the points along the path of the corner homing 45
    # point0 is the point where they touched
    def get_corner_homing_45_pathpoints(point0):
      p0x = point0[0]
      p0y = point0[1]
      p0z = point0[2]
      p0rx = point0[3]
      p0ry = point0[4]
      p0rz = point0[5]

      #constants
      #distances of how far away from point the touchpoints are
      d0 = 0.15 # how far from the box to retreat and approach
      d1 = 0.05
      d2 = 0.2
      sqrt2 = 0.707106781

      ph1 = p[p0x + d0, p0y, p0z + .05, p0rx, p0ry, p0rz] #approach point for turn

      ph2 = p[p0x+d0-d0*sqrt2-sqrt2*d1, p0y+d0*sqrt2+sqrt2*d1, p0z+.05, .445, -1.562, .483]
      ph3 = p[p0x+d0-d0*sqrt2-sqrt2*d2, p0y+d0*sqrt2+sqrt2*d2, p0z+.05, .445, -1.562, .483]
      ph4 = p[p0x+d0-d0*sqrt2-sqrt2*d1, p0y-d0*sqrt2-sqrt2*d1, p0z+.05, 1.699, 3.576, 1.841]
      ph5 = p[p0x+d0-d0*sqrt2-sqrt2*d2, p0y-d0*sqrt2-sqrt2*d2, p0z+.05, 1.699, 3.576, 1.841]

      # go back to ph1
      ph6 = p[p0x + .05, p0y, p0z -.05, 0, 0, 0] # approach point for under turn
      # moveL from ph1 to ph6
      ph7 = p[p0x-.05, p0y, p0z-.05, 0, 0, 0]
      ret = struct(ph1=ph1, ph2=ph2, ph3=ph3, ph4=ph4, ph5=ph5, ph6=ph6, ph7=ph7)
      return ret
    end
    $ 203 "path_pre≔get_corner_homing_45_pathpoints(tp)"
    global path_pre=get_corner_homing_45_pathpoints(tp)
    $ 204 "ph1≔path_pre[0]"
    global ph1=path_pre[0]
    $ 205 "ph2≔path_pre[1]"
    global ph2=path_pre[1]
    $ 206 "ph3≔path_pre[2]"
    global ph3=path_pre[2]
    $ 207 "ph4≔path_pre[3]"
    global ph4=path_pre[3]
    $ 208 "ph5≔path_pre[4]"
    global ph5=path_pre[4]
    $ 209 "ph6≔path_pre[5]"
    global ph6=path_pre[5]
    $ 210 "ph7≔path_pre[6]"
    global ph7=path_pre[6]
    $ 211 "MoveJ"
    $ 212 "ph1" "breakAfter"
    movej(ph1, a=1.3962634015954636, v=1.0471975511965976)
    $ 213 "ph2" "breakAfter"
    movej(ph2, a=1.3962634015954636, v=1.0471975511965976)
    $ 214 "MoveL"
    $ 215 "Direction: Base"
    global move_thread_flag_215=0
    thread move_thread_215():
      enter_critical
      move_thread_flag_215 = 1
      local towardsPos=calculate_point_to_move_towards(p[0.0,0.0,0.0,0.0,0.0,0.0], [-1,-1.0,0.0], 1000.0)
      movel(towardsPos, a=0.1, v=0.05)
      move_thread_flag_215 = 2
      exit_critical
    end
    move_thread_flag_215 = 0
    move_thread_han_215 = run move_thread_215()
    while (True):
      local targetTcpDirection=get_target_tcp_speed()
      local stepsToRetract=tool_contact(direction=targetTcpDirection)
      if (stepsToRetract > 0):
        kill move_thread_han_215
        stopl(3.0)
        local backTrackMovement=get_actual_joint_positions_history(stepsToRetract)
        local contactPose=get_forward_kin(backTrackMovement)
        local posDir=[targetTcpDirection[0],targetTcpDirection[1],targetTcpDirection[2]]
        local retractTo=contactPose
        if (norm(posDir) > 1e-6):
          local normalizedPosDir=normalize(posDir)
          local additionalRetraction=p[normalizedPosDir[0] * 0.0, normalizedPosDir[1] * 0.0, normalizedPosDir[2] * 0.0, 0, 0, 0]
          retractTo = pose_sub(contactPose, additionalRetraction)
        end
        movel(retractTo, a=3.0, v=0.1)
        $ 216 "Until (tool_contact_detection)"
        break
      end
      sync()
    end
    $ 217 "p11≔get_actual_tcp_pose()"
    global p11= get_actual_tcp_pose ()
    $ 218 "MoveJ"
    $ 219 "ph3" "breakAfter"
    movej(ph3, a=1.3962634015954636, v=1.0471975511965976)
    $ 220 "MoveL"
    $ 221 "Direction: Base"
    global move_thread_flag_221=0
    thread move_thread_221():
      enter_critical
      move_thread_flag_221 = 1
      local towardsPos=calculate_point_to_move_towards(p[0.0,0.0,0.0,0.0,0.0,0.0], [-1,-1.0,0.0], 1000.0)
      movel(towardsPos, a=0.1, v=0.05)
      move_thread_flag_221 = 2
      exit_critical
    end
    move_thread_flag_221 = 0
    move_thread_han_221 = run move_thread_221()
    while (True):
      local targetTcpDirection=get_target_tcp_speed()
      local stepsToRetract=tool_contact(direction=targetTcpDirection)
      if (stepsToRetract > 0):
        kill move_thread_han_221
        stopl(3.0)
        local backTrackMovement=get_actual_joint_positions_history(stepsToRetract)
        local contactPose=get_forward_kin(backTrackMovement)
        local posDir=[targetTcpDirection[0],targetTcpDirection[1],targetTcpDirection[2]]
        local retractTo=contactPose
        if (norm(posDir) > 1e-6):
          local normalizedPosDir=normalize(posDir)
          local additionalRetraction=p[normalizedPosDir[0] * 0.0, normalizedPosDir[1] * 0.0, normalizedPosDir[2] * 0.0, 0, 0, 0]
          retractTo = pose_sub(contactPose, additionalRetraction)
        end
        movel(retractTo, a=3.0, v=0.1)
        $ 222 "Until (tool_contact_detection)"
        break
      end
      sync()
    end
    $ 223 "p12≔get_actual_tcp_pose()"
    global p12= get_actual_tcp_pose ()
    $ 224 "MoveJ"
    $ 225 "ph3" "breakAfter"
    movej(ph3, a=1.3962634015954636, v=1.0471975511965976)
    $ 226 "Waypoint_10" "breakAfter"
    movej(get_inverse_kin(Waypoint_10_p, qnear=Waypoint_10_q), a=1.3962634015954636, v=1.0471975511965976)
    $ 227 "MoveJ"
    $ 228 "Waypoint_11" "breakAfter"
    movej(get_inverse_kin(Waypoint_11_p, qnear=Waypoint_11_q), a=1.3962634015954636, v=1.0471975511965976)
    $ 230 "Waypoint_12" "breakAfter"
    movej(get_inverse_kin(Waypoint_12_p, qnear=Waypoint_12_q), a=1.3962634015954636, v=1.0471975511965976)
    $ 231 "MoveJ"
    $ 232 "ph4" "breakAfter"
    movej(ph4, a=1.3962634015954636, v=1.0471975511965976)
    $ 233 "MoveL"
    $ 234 "Direction: Base"
    global move_thread_flag_234=0
    thread move_thread_234():
      enter_critical
      move_thread_flag_234 = 1
      local towardsPos=calculate_point_to_move_towards(p[0.0,0.0,0.0,0.0,0.0,0.0], [-1.0,1.0,0.0], 1000.0)
      movel(towardsPos, a=0.1, v=0.05)
      move_thread_flag_234 = 2
      exit_critical
    end
    move_thread_flag_234 = 0
    move_thread_han_234 = run move_thread_234()
    while (True):
      local targetTcpDirection=get_target_tcp_speed()
      local stepsToRetract=tool_contact(direction=targetTcpDirection)
      if (stepsToRetract > 0):
        kill move_thread_han_234
        stopl(3.0)
        local backTrackMovement=get_actual_joint_positions_history(stepsToRetract)
        local contactPose=get_forward_kin(backTrackMovement)
        local posDir=[targetTcpDirection[0],targetTcpDirection[1],targetTcpDirection[2]]
        local retractTo=contactPose
        if (norm(posDir) > 1e-6):
          local normalizedPosDir=normalize(posDir)
          local additionalRetraction=p[normalizedPosDir[0] * 0.0, normalizedPosDir[1] * 0.0, normalizedPosDir[2] * 0.0, 0, 0, 0]
          retractTo = pose_sub(contactPose, additionalRetraction)
        end
        movel(retractTo, a=3.0, v=0.1)
        $ 235 "Until (tool_contact_detection)"
        break
      end
      sync()
    end
    $ 236 "p21≔get_actual_tcp_pose()"
    global p21= get_actual_tcp_pose ()
    $ 237 "MoveJ"
    $ 238 "ph5" "breakAfter"
    movej(ph5, a=1.3962634015954636, v=1.0471975511965976)
    $ 239 "MoveL"
    $ 240 "Direction: Base"
    global move_thread_flag_240=0
    thread move_thread_240():
      enter_critical
      move_thread_flag_240 = 1
      local towardsPos=calculate_point_to_move_towards(p[0.0,0.0,0.0,0.0,0.0,0.0], [-1.0,1.0,0.0], 1000.0)
      movel(towardsPos, a=0.1, v=0.05)
      move_thread_flag_240 = 2
      exit_critical
    end
    move_thread_flag_240 = 0
    move_thread_han_240 = run move_thread_240()
    while (True):
      local targetTcpDirection=get_target_tcp_speed()
      local stepsToRetract=tool_contact(direction=targetTcpDirection)
      if (stepsToRetract > 0):
        kill move_thread_han_240
        stopl(3.0)
        local backTrackMovement=get_actual_joint_positions_history(stepsToRetract)
        local contactPose=get_forward_kin(backTrackMovement)
        local posDir=[targetTcpDirection[0],targetTcpDirection[1],targetTcpDirection[2]]
        local retractTo=contactPose
        if (norm(posDir) > 1e-6):
          local normalizedPosDir=normalize(posDir)
          local additionalRetraction=p[normalizedPosDir[0] * 0.0, normalizedPosDir[1] * 0.0, normalizedPosDir[2] * 0.0, 0, 0, 0]
          retractTo = pose_sub(contactPose, additionalRetraction)
        end
        movel(retractTo, a=3.0, v=0.1)
        $ 241 "Until (tool_contact_detection)"
        break
      end
      sync()
    end
    $ 242 "p22≔get_actual_tcp_pose()"
    global p22= get_actual_tcp_pose ()
    $ 243 "MoveJ"
    $ 244 "ph5" "breakAfter"
    movej(ph5, a=1.3962634015954636, v=1.0471975511965976)
    $ 245 "ph4" "breakAfter"
    movej(ph4, a=1.3962634015954636, v=1.0471975511965976)
    $ 247 "Waypoint_13" "breakAfter"
    movej(get_inverse_kin(Waypoint_13_p, qnear=Waypoint_13_q), a=1.3962634015954636, v=1.0471975511965976)
    $ 248 "Waypoint_14" "breakAfter"
    movej(get_inverse_kin(Waypoint_14_p, qnear=Waypoint_14_q), a=1.3962634015954636, v=1.0471975511965976)
    $ 249 "Waypoint_15" "breakAfter"
    movej(get_inverse_kin(Waypoint_15_p, qnear=Waypoint_15_q), a=1.3962634015954636, v=1.0471975511965976)
    $ 250 "Waypoint_16" "breakAfter"
    movej(get_inverse_kin(Waypoint_16_p, qnear=Waypoint_16_q), a=1.3962634015954636, v=1.0471975511965976)
    $ 251 "ph6" "breakAfter"
    movej(ph6, a=1.3962634015954636, v=1.0471975511965976)
    $ 252 "ph7" "breakAfter"
    movej(ph7, a=1.3962634015954636, v=1.0471975511965976)
    $ 253 "MoveL"
    $ 254 "Direction: Base Z+"
    global move_thread_flag_254=0
    thread move_thread_254():
      enter_critical
      move_thread_flag_254 = 1
      local towardsPos=calculate_point_to_move_towards(p[0.0,0.0,0.0,0.0,0.0,0.0], [0.0,0.0,1.0], 1000.0)
      movel(towardsPos, a=0.1, v=0.05)
      move_thread_flag_254 = 2
      exit_critical
    end
    move_thread_flag_254 = 0
    move_thread_han_254 = run move_thread_254()
    while (True):
      local targetTcpDirection=get_target_tcp_speed()
      local stepsToRetract=tool_contact(direction=targetTcpDirection)
      if (stepsToRetract > 0):
        kill move_thread_han_254
        stopl(3.0)
        local backTrackMovement=get_actual_joint_positions_history(stepsToRetract)
        local contactPose=get_forward_kin(backTrackMovement)
        local posDir=[targetTcpDirection[0],targetTcpDirection[1],targetTcpDirection[2]]
        local retractTo=contactPose
        if (norm(posDir) > 1e-6):
          local normalizedPosDir=normalize(posDir)
          local additionalRetraction=p[normalizedPosDir[0] * 0.0, normalizedPosDir[1] * 0.0, normalizedPosDir[2] * 0.0, 0, 0, 0]
          retractTo = pose_sub(contactPose, additionalRetraction)
        end
        movel(retractTo, a=3.0, v=0.1)
        $ 255 "Until (tool_contact_detection)"
        break
      end
      sync()
    end
    $ 256 "p3≔get_actual_tcp_pose()"
    global p3= get_actual_tcp_pose ()
    $ 257 "MoveJ"
    $ 258 "ph7" "breakAfter"
    movej(ph7, a=1.3962634015954636, v=1.0471975511965976)
    $ 259 "ph6" "breakAfter"
    movej(ph6, a=1.3962634015954636, v=1.0471975511965976)
    $ 260 "Waypoint_17" "breakAfter"
    movej(get_inverse_kin(Waypoint_17_p, qnear=Waypoint_17_q), a=1.3962634015954636, v=1.0471975511965976)
    $ 261 "Waypoint_18" "breakAfter"
    movej(get_inverse_kin(Waypoint_18_p, qnear=Waypoint_18_q), a=1.3962634015954636, v=1.0471975511965976)
    $ 262 "Home"
    movej([-3.4579734502641006, -2.05691362454537, 2.326567589830591, -0.22707360390354125, -0.19934432301767302, -0.10534790278823536], a=1.3962634015954636, v=1.0471975511965976)
    $ 263 "Comment"
    # Comment
    $ 264 "Comment"
    # Comment
    $ 265 "Comment"
    # Comment
    $ 266 "Comment"
    # Comment
    $ 267 "Comment"
    # Comment
    $ 268 "Comment"
    # Comment
  end
  $ 269 "Thread_1"
  thread Thread_1():
    while (True):
      $ 270 "Loop  True "
      while (  True  ):
        $ 271 "If freedrive_m_var≟ True "
        if (freedrive_m_var ==   True  ):
          $ 272 "freedrive_mode()"
          freedrive_mode()
        else:
          $ 273 "Else" "noBreak"
          $ 274 "end_freedrive_mode()"
          end_freedrive_mode()
        end
        $ 275 "sync()"
        sync()
      end
    end
  end
  threadId_Thread_1 = run Thread_1()
  $ 276 "Thread_2"
  thread Thread_2():
    while (True):
      $ 277 "Loop  True "
      while (  True  ):
        $ 278 "If thread2trigger≟ True "
        if (thread2trigger ==   True  ):
          $ 279 "'do the dot extrude'"
          # 'do the dot extrude'
          $ 280 "Wait: 5.0"
          sleep(5.0)
          # begin: URCap Program Node
          #   Source: WireTank Serial, 4.8.0, WireTank, LLC
          #   Type: WireTank Serial
          $ 281 "Serial Bridge uR1"
          SerialResponse = WTSerialBridge.send_command("/dev/ttyUSB0",1200, 8, "None", "One", "None", 5000, "None", "None", [252,82,49], False)
          # end: URCap Program Node
          $ 282 "Wait: 2.0"
          sleep(2.0)
          # begin: URCap Program Node
          #   Source: WireTank Serial, 4.8.0, WireTank, LLC
          #   Type: WireTank Serial
          $ 283 "Serial Bridge uR0"
          SerialResponse = WTSerialBridge.send_command("/dev/ttyUSB0",1200, 8, "None", "One", "None", 5000, "None", "None", [252,82,48], False)
          # end: URCap Program Node
          $ 284 "thread2trigger≔ False "
          global thread2trigger=  False
        end
        $ 285 "sync()"
        sync()
      end
    end
  end
  threadId_Thread_2 = run Thread_2()
  $ 2 "Robot Program"
  $ 3 "'start of main program'"
  # 'start of main program'
  $ 4 "Home"
  movej([-3.4579734502641006, -2.05691362454537, 2.326567589830591, -0.22707360390354125, -0.19934432301767302, -0.10534790278823536], a=1.3962634015954636, v=1.0471975511965976)
  $ 5 "Set"
  set_tcp(p[0.00157,-0.09008,0.25767,0.0,0.0,0.0])
  $ 6 "Test_Teach_Position()"
  Test_Teach_Position()
  $ 7 "Set"
  set_tcp(p[0.00157,-0.09008,0.25767,0.0,0.0,0.0])
  $ 8 "Corner_Homing_45()"
  Corner_Homing_45()
  $ 9 "Set"
  set_tcp(p[-0.00438,-0.33062,0.10207,1.2092,-1.2092,1.2092])
  $ 10 "extrude_knife2()"
  extrude_knife2()
  $ 11 "Script: analyze_touchpoints.script"
  # this file creates the function for analyzing touchpoints
  # define pi
  pi = 3.1415926535

  # this is the main entry point for calculations.
  # it takes in the 5 points, analyzes the shape of the box, and then calculates path points and returns them
  # specifically for Down, Over, then Around (DOtA)
  # specifically for right-sided boxes (vertical weld on right side of edge)
  def main_calculate_right(p11, p12, p21, p22, p3):
      struct1 = analyze_touchpoints_only(p11, p12, p21, p22, p3)
      struct2 = calculate_DOtA_points_right(struct1)
      return struct2
  end

  # this is the main entry point for calculations.
  # it takes in the 5 points, analyzes the shape of the box, and then calculates path points and returns them
  # specifically for Down, Over, then Around (DOtA)
  # specifically for left-sided boxes (vertical weld on left side of edge)
  def main_calculate_left(p11, p12, p21, p22, p3):
      struct1 = analyze_touchpoints_only(p11, p12, p21, p22, p3)
      struct2 = calculate_DOtA_points_left(struct1)
      return struct2
  end

  # it takes 5 arguments as points
  # it returns a struct containing: (pointintersect, pointapproach1, pointapproach2, point1, point2, point3, point4, point5, pointreturn1, heading1, heading2, heading3, path2r1, path2r2, path2l1, path2l2)
  # specifically for Around then Up (AtU)
  def analyze_touchpoints(p11, p12, p21, p22, p3):
    # FIND THE INTERSECTION
    # comment get the z
    zcoord=p3[2]

    # get the raw points from the first line
    l1p1x=p11[0]
    l1p1y=p11[1]
    l1p2x=p12[0]
    l1p2y=p12[1]

    # equate the first line in 2d space
    ml1 = (l1p2y-l1p1y) / (l1p2x-l1p1x)

    # b = y - mx
    bl1 = l1p1y - ml1 * l1p1x

    # get the raw points from the second line
    l2p1x=p21[0]
    l2p1y=p21[1]
    l2p2x=p22[0]
    l2p2y=p22[1]

    # equate the second line in 2d space
    ml2 = (l2p2y-l2p1y) / (l2p2x-l2p1x)

    # b = y - mx
    bl2 = l2p1y - ml2 * l2p1x


    # find the intersection of the two lines
    # m1x+b1 = m2x+b2
    # m1x - m2x = b2 - b1
    # x = (b2-b1) / (m1-m2)
    xintersect = (bl2-bl1) / (ml1-ml2)
    yintersect = ml1 * xintersect + bl1

    #FIND THE VECTORS
    #define a vector from the intersection to the second point on the first line
    l1delxfull = l1p2x - xintersect
    l1delyfull = l1p2y - yintersect

    l1delmag = sqrt(l1delxfull*l1delxfull + l1delyfull*l1delyfull)

    l1delxunit = l1delxfull / l1delmag
    l1delyunit = l1delyfull / l1delmag

    #define a vector from the intersection to the second point on the second line
    l2delxfull = l2p2x - xintersect
    l2delyfull = l2p2y - yintersect

    l2delmag = sqrt(l2delxfull*l2delxfull + l2delyfull*l2delyfull)

    l2delxunit = l2delxfull / l2delmag
    l2delyunit = l2delyfull / l2delmag

    # FIND THE FOUR POINTS ON THE LINES
    # find locations 8 inches away from  intersect point
    # CONST
    welddistance = 8
    roundoverdistance = 0.05
    zup = .375
    # inches
    wd = welddistance * 25.4 / 1000
    rod = roundoverdistance * 25.4 / 1000
    zup = zup * 25.4 / 1000

    # now we have the unit vector. extend the weld distance from the intersection
    x = xintersect + l1delxunit * wd
    y = yintersect + l1delyunit * wd
    z = zcoord + zup

    point1 = p[x,y,z,1.570796,0,0] # dummy orientation for now

    x = xintersect + l1delxunit * rod
    y = yintersect + l1delyunit * rod

    point2 = p[x,y,z,1.570796,0,0]

    # now we have the unit vector. extend the weld distance from the intersection
    x = xintersect + l2delxunit * wd
    y = yintersect + l2delyunit * wd

    point5 = p[x,y,z,0,-1.570796,0]

    x = xintersect + l2delxunit * rod
    y = yintersect + l2delyunit * rod

    point4 = p[x,y,z,0,-1.570796,0]

    #DEFINE APPROACH POINTS
    pointintersect = p[xintersect,yintersect,zcoord,0,0,0]
    pointapproach1 = p[xintersect+0.1,yintersect+0.1,z,1.570796,0,0]
    pointapproach2 = p[point1[0], point1[1]+0.1, point1[2], point1[3], point1[4], point1[5]]
    pointreturn1 = p[point5[0]+0.1, point5[1], point5[2], point5[3], point5[4], point5[5]]

    #FIND HEADINGS
    #for each heading, find the angle of the line with respect to the pos x axis. then add/subtract 90 degrees because you want to be perpendicular to that
    headingvector1 = convert_uv_to_heading(l1delxunit, l1delyunit)
    headingvector2 = convert_uv_to_heading(l2delxunit, l2delyunit)
    # find halfway heading
    heading2 = (headingvector1 + headingvector2)/2
    # find headings that the robot should face while traveling, perpendicular to the vectors of the sides of the box
    heading1 = headingvector1 + pi/2
    heading3 = headingvector2 - pi/2

    #FIND POINT 3
    #see if we have to / can find point 3
    findpoint3 = True
    if roundoverdistance == 0:
      findpoint3 = False
    end
    if findpoint3:
      # i need to find the point3 such that the arc from p2 to p3 to p4 is tangent to p1-p2 and p4-p5. making this a smooth path will be good
      # the direction of movement is from pointintersect in the direction of heading2
      # how much movement though? this will depend on whether it is actually a 90 degree angle or not.
      # first, find the perpendicular lines through points 2 and 4
      perp2 = find_perpendicular_line(ml1, point2[0], point2[1])
      perp4 = find_perpendicular_line(ml2, point4[0], point4[1])
      # next, find the intersection of those two lines
      perpintersect = find_intersection(perp2[0], perp2[1], perp4[0], perp4[1])
      radiusofcircle = distance_between(perpintersect[0], perpintersect[1], 0, point2[0], point2[1], 0)
      # find a vector the direction of heading2
      uvx = cos(heading2)
      uvy = sin(heading2)
      # compute point3. pass in negative radius because the direction is into the tank but we want to move from the intersection out to the rounded edge.
      point3coords = add_vectordistance_to_point(perpintersect[0], perpintersect[1], z, uvx, uvy, 0, -1 * radiusofcircle)
      point3 = p[point3coords[0], point3coords[1], point3coords[2], 0, 0, 0]
    end

    #APPLY ACTUAL RXRYRZ TO POINTS
    # convert the headings to rxryrz and insert those values into the relevant points
    rxryrz = convert_heading_to_axang(heading1)
    rx = rxryrz[0]
    ry = rxryrz[1]
    rz = rxryrz[2]
    pointapproach1 = p[pointapproach1[0], pointapproach1[1], pointapproach1[2], rx, ry, rz]
    pointapproach2 = p[pointapproach2[0], pointapproach2[1], pointapproach2[2], rx, ry, rz]
    point1 = p[point1[0], point1[1], point1[2], rx, ry, rz]
    point2 = p[point2[0], point2[1], point2[2], rx, ry, rz]
    rxryrz = convert_heading_to_axang(heading2)
    rx = rxryrz[0]
    ry = rxryrz[1]
    rz = rxryrz[2]
    if findpoint3:
      point3 = p[point3[0], point3[1], point3[2], rx, ry, rz]
    else:
      point3 = point2
    end
    rxryrz = convert_heading_to_axang(heading3)
    rx = rxryrz[0]
    ry = rxryrz[1]
    rz = rxryrz[2]
    point4 = p[point4[0], point4[1], point4[2], rx, ry, rz]
    point5 = p[point5[0], point5[1], point5[2], rx, ry, rz]
    pointreturn1 = p[pointreturn1[0], pointreturn1[1], pointreturn1[2], rx, ry, rz]

    #find path2 (the part that goes up)
    four_vertical_points = find_vertical_points(pointintersect, l1delxunit, l1delyunit, l2delxunit, l2delyunit, zup, wd, heading1, heading3)
    path2r1 = four_vertical_points[0]
    path2r2 = four_vertical_points[1]
    path2l1 = four_vertical_points[2]
    path2l2 = four_vertical_points[3]

    #RETURN STRUCT
    ret = struct(pointintersect=pointintersect, pointapproach1=pointapproach1, pointapproach2=pointapproach2, point1=point1, point2=point2, point3=point3, point4=point4, point5=point5, pointreturn1=pointreturn1, heading1=heading1, heading2=heading2, heading3=heading3, path2r1=path2r1, path2r2=path2r2, path2l1=path2l1, path2l2=path2l2)
    return ret
  end

  # it takes 5 arguments as points
  # it returns a struct containing: (pointintersect, heading1, heading2, heading3, l1delxunit, l1delyunit, l2delxunit, l2delyunit)
  def analyze_touchpoints_only(p11, p12, p21, p22, p3):
    # FIND THE INTERSECTION
    # comment get the z
    zcoord=p3[2]

    # get the raw points from the first line
    l1p1x=p11[0]
    l1p1y=p11[1]
    l1p2x=p12[0]
    l1p2y=p12[1]

    # equate the first line in 2d space
    ml1 = (l1p2y-l1p1y) / (l1p2x-l1p1x)

    # b = y - mx
    bl1 = l1p1y - ml1 * l1p1x

    # get the raw points from the second line
    l2p1x=p21[0]
    l2p1y=p21[1]
    l2p2x=p22[0]
    l2p2y=p22[1]

    # equate the second line in 2d space
    ml2 = (l2p2y-l2p1y) / (l2p2x-l2p1x)

    # b = y - mx
    bl2 = l2p1y - ml2 * l2p1x


    # find the intersection of the two lines
    # m1x+b1 = m2x+b2
    # m1x - m2x = b2 - b1
    # x = (b2-b1) / (m1-m2)
    xintersect = (bl2-bl1) / (ml1-ml2)
    yintersect = ml1 * xintersect + bl1

    pointintersect = p[xintersect,yintersect,zcoord,0,0,0]

    #FIND THE VECTORS
    #define a vector from the intersection to the second point on the first line
    l1delxfull = l1p2x - xintersect
    l1delyfull = l1p2y - yintersect

    l1delmag = sqrt(l1delxfull*l1delxfull + l1delyfull*l1delyfull)

    l1delxunit = l1delxfull / l1delmag
    l1delyunit = l1delyfull / l1delmag

    #define a vector from the intersection to the second point on the second line
    l2delxfull = l2p2x - xintersect
    l2delyfull = l2p2y - yintersect

    l2delmag = sqrt(l2delxfull*l2delxfull + l2delyfull*l2delyfull)

    l2delxunit = l2delxfull / l2delmag
    l2delyunit = l2delyfull / l2delmag

    #FIND HEADINGS
    #for each heading, find the angle of the line with respect to the pos x axis. then add/subtract 90 degrees because you want to be perpendicular to that
    headingvector1 = convert_uv_to_heading(l1delxunit, l1delyunit)
    headingvector2 = convert_uv_to_heading(l2delxunit, l2delyunit)
    # find halfway heading
    heading2 = (headingvector1 + headingvector2)/2
    # find headings that the robot should face while traveling, perpendicular to the vectors of the sides of the box
    heading1 = headingvector1 + pi/2
    heading3 = headingvector2 - pi/2

    #RETURN STRUCT
    ret = struct(pointintersect=pointintersect, heading1=heading1, heading2=heading2, heading3=heading3, l1delxunit=l1delxunit, l1delyunit=l1delyunit, l2delxunit=l2delxunit, l2delyunit=l2delyunit)
    return ret
  end

  # given a struct from analyze_touchpoints_only(), calculate the points
  def calculate_DOtA_points_right(struct1):
      # get the stuff from the struct
      pointintersect = struct1[0]
      heading1 = struct1[1]
      heading2 = struct1[2]
      heading3 = struct1[3]
      l1delxunit = struct1[4]
      l1delyunit = struct1[5]
      l2delxunit = struct1[6]
      l2delyunit = struct1[7]

      # FIND THE POINTS ON THE LINES OF THE FIRST TURN PATH
      # find locations 8 inches away from  intersect point
      # CONST
      welddistance1 = 8 # vertical weld distance
      welddistance2 = 3 # first path second leg
      welddistance3 = 8 # second path second leg
      zup = .375
      # inches
      wd1 = welddistance1 * 25.4 / 1000
      wd2 = welddistance2 * 25.4 / 1000
      wd3 = welddistance3 * 25.4 / 1000
      zup = zup * 25.4 / 1000

      x = pointintersect[0] + l1delxunit * zup
      y = pointintersect[1] + l1delyunit * zup
      z = pointintersect[2] + zup

      #apply actual rxryrz to points
      # convert the headings to rxryrz and insert those values into the relevant points
      rxryrz = convert_heading_to_axang_preheatdown(heading1)
      rx = rxryrz[0]
      ry = rxryrz[1]
      rz = rxryrz[2]

      point1 = p[x, y, z + wd1, rx, ry, rz]
      point2 = p[x, y, z, rx, ry, rz]

      # convert the headings to rxryrz and insert those values into the relevant points
      rxryrz = convert_heading_to_axang_ccw(heading1)
      rx = rxryrz[0]
      ry = rxryrz[1]
      rz = rxryrz[2]

      point4 = p[x, y, z, rx, ry, rz]
      x = x + l1delxunit * wd2
      y = y + l1delyunit * wd2
      point5 = p[x, y, z, rx, ry, rz]

      # FIND THE POINTS ON THE LINES OF THE SECOND AROUND PATH
      roundoverdistance = 0.05
      rod = roundoverdistance * 25.4 / 1000

      # now we have the unit vector. extend the weld distance from the intersection
      x = pointintersect[0] + l1delxunit * (zup)
      y = pointintersect[1] + l1delyunit * zup
      # convert the headings to rxryrz and insert those values into the relevant points
      rxryrz = convert_heading_to_axang(heading1)
      rx = rxryrz[0]
      ry = rxryrz[1]
      rz = rxryrz[2]
      point_1 = p[x, y, z, rx, ry, rz]

      x = pointintersect[0] + l1delxunit * rod
      y = pointintersect[1] + l1delyunit * rod
      point_2 = p[x, y, z, rx, ry, rz]

      # now we have the unit vector. extend the weld distance from the intersection
      x = pointintersect[0] + l2delxunit * wd3
      y = pointintersect[1] + l2delyunit * wd3
      # convert the headings to rxryrz and insert those values into the relevant points
      rxryrz = convert_heading_to_axang(heading3)
      rx = rxryrz[0]
      ry = rxryrz[1]
      rz = rxryrz[2]
      point_5 = p[x, y, z, rx, ry, rz]

      x = pointintersect[0] + l2delxunit * rod
      y = pointintersect[1] + l2delyunit * rod
      point_4 = p[x, y, z, rx, ry, rz]

      #FIND POINT 3
      # by calling analyze_touchpoints()
      atret = analyze_touchpoints(point_2, point_1, point_4, point_5, pointintersect)
      point_3 = atret[5]


      struct2 = struct(point1=point1, point2=point2, point4=point4, point5=point5, point_1=point_1, point_2=point_2, point_3=point_3, point_4=point_4, point_5=point_5)
      return struct2
  end

  # given a struct from analyze_touchpoints_only(), calculate the points
  def calculate_DOtA_points_left(struct1):
      # get the stuff from the struct
      pointintersect = struct1[0]
      heading1 = struct1[1]
      heading2 = struct1[2]
      heading3 = struct1[3]
      l1delxunit = struct1[4]
      l1delyunit = struct1[5]
      l2delxunit = struct1[6]
      l2delyunit = struct1[7]

      # FIND THE POINTS ON THE LINES OF THE FIRST TURN PATH
      # find locations 8 inches away from  intersect point
      # CONST
      welddistance = 8
      zup = .375
      # inches
      wd = welddistance * 25.4 / 1000
      zup = zup * 25.4 / 1000

      x = pointintersect[0] + l2delxunit * zup
      y = pointintersect[1] + l2delyunit * zup
      z = pointintersect[2] + zup

      #apply actual rxryrz to points
      # convert the headings to rxryrz and insert those values into the relevant points
      rxryrz = convert_heading_to_axang_preheatdown(heading3)
      rx = rxryrz[0]
      ry = rxryrz[1]
      rz = rxryrz[2]

      point1 = p[x, y, z + wd, rx, ry, rz]
      point2 = p[x, y, z, rx, ry, rz]

      # convert the headings to rxryrz and insert those values into the relevant points
      rxryrz = convert_heading_to_axang(heading3)
      rx = rxryrz[0]
      ry = rxryrz[1]
      rz = rxryrz[2]

      point4 = p[x, y, z, rx, ry, rz]
      x = x + l2delxunit * wd
      y = y + l2delyunit * wd
      point5 = p[x, y, z, rx, ry, rz]

      # FIND THE POINTS ON THE LINES OF THE SECOND AROUND PATH
      roundoverdistance = 0.05
      rod = roundoverdistance * 25.4 / 1000

      # now we have the unit vector. extend the weld distance from the intersection
      x = pointintersect[0] + l2delxunit * (zup)
      y = pointintersect[1] + l2delyunit * zup
      # convert the headings to rxryrz and insert those values into the relevant points
      rxryrz = convert_heading_to_axang_ccw(heading3)
      rx = rxryrz[0]
      ry = rxryrz[1]
      rz = rxryrz[2]
      point_1 = p[x, y, z, rx, ry, rz]

      x = pointintersect[0] + l2delxunit * rod
      y = pointintersect[1] + l2delyunit * rod
      point_2 = p[x, y, z, rx, ry, rz]

      # now we have the unit vector. extend the weld distance from the intersection
      x = pointintersect[0] + l1delxunit * wd
      y = pointintersect[1] + l1delyunit * wd
      # convert the headings to rxryrz and insert those values into the relevant points
      rxryrz = convert_heading_to_axang_ccw(heading1)
      rx = rxryrz[0]
      ry = rxryrz[1]
      rz = rxryrz[2]
      point_5 = p[x, y, z, rx, ry, rz]

      x = pointintersect[0] + l1delxunit * rod
      y = pointintersect[1] + l1delyunit * rod
      point_4 = p[x, y, z, rx, ry, rz]

      #FIND POINT 3
      # by calling analyze_touchpoints()
      atret = analyze_touchpoints(point_2, point_1, point_4, point_5, pointintersect)
      point_3 = atret[5]
      #point 3 will not have the correct rxryrz though because now the gun needs to be face up.
      rxryrz = convert_heading_to_axang_ccw(heading2)
      rx = rxryrz[0]
      ry = rxryrz[1]
      rz = rxryrz[2]
      point_3 = p[point_3[0], point_3[1], point_3[2], rx, ry, rz]

      struct2 = struct(point1=point1, point2=point2, point4=point4, point5=point5, point_1=point_1, point_2=point_2, point_3=point_3, point_4=point_4, point_5=point_5)
      return struct2
  end

  # given a heading, (ccw from +x axis), find the mx+b slope
  # fails if exactly vertical
  def get_slope_from_heading(heading):
      return tan(heading)
  end



  # this function finds the points (and rxryrz) of the 2 points (start and end) of vertical weld section
  def find_vertical_points(pointintersect, l1delxunit, l1delyunit, l2delxunit, l2delyunit, offset, wd, heading1, heading3):

    # find right side stuff
    # find the point in 3d space that is .375 up and .375 over
    x = pointintersect[0] + l1delxunit * offset
    y = pointintersect[1] + l1delyunit * offset
    z = pointintersect[2] + offset
    # find rxryrz
    rxryrz = convert_heading_to_axang_preheatup(heading1)
    rx = rxryrz[0]
    ry = rxryrz[1]
    rz = rxryrz[2]
    path2r1 = p[x, y, z, rx, ry, rz]
    path2r2 = p[x, y, z + wd, rx, ry, rz]

    # find left side
    # find the point in 3d space that is .375 up and .375 over
    x = pointintersect[0] + l2delxunit * offset
    y = pointintersect[1] + l2delyunit * offset
    z = pointintersect[2] + offset
    # find rxryrz
    rxryrz = convert_heading_to_axang_preheatup(heading3)
    rx = rxryrz[0]
    ry = rxryrz[1]
    rz = rxryrz[2]
    path2l1 = p[x, y, z, rx, ry, rz]
    path2l2 = p[x, y, z + wd, rx, ry, rz]

    ret = struct(path2r1=path2r1, path2r2=path2r2, path2l1=path2l1, path2l2=path2l2)
    return ret
  end

  # this function converts a unit vector to its heading angle ccw from x+ axis
  # takes uvx and uvy
  # returns heading in radians
  def convert_uv_to_heading(uvx, uvy):
    baseang = atan(uvy/uvx)
    if uvx < 0:
      ang = baseang + pi
    elif uvy < 0:
      ang = baseang + pi * 2
    else:
      ang = baseang
    end
    return ang
  end

  # this function finds the equation of a line, perpendicular to a given line, and going through a given point
  # takes 3 arguments: m (the original line's slope), x (point's x coord), y (point's y coord). the b of the original line is not needed
  # returns a list of [m,b] (the slope and intercept of the new line)
  def find_perpendicular_line(origm, x, y):
    m = (1/origm) * -1
    b = y - m*x
    ret = [m, b]
    return ret
  end

  # this function finds the intersection point between two lines in the xy plane
  # takes 4 arguments: m1, b1, m2, b2
  # returns a list of [x,y] (the point of intersection)
  def find_intersection(m1, b1, m2, b2):
    # m1x+b1 = m2x+b2
    # m1x - m2x = b2 - b1
    # x = (b2-b1) / (m1-m2)
    x = (b2-b1) / (m1-m2)
    y = m1 * x + b1
    ret = [x, y]
    return ret
  end

  # this function finds the distance between 2 points in 3d space
  # it takes 6 arguments: x1, y1, z1, x2, y2, z2
  # it returns a distance
  def distance_between(x1, y1, z1, x2, y2, z2):
    distsquared = (x2-x1)*(x2-x1)+(y2-y1)*(y2-y1)+(z2-z1)*(z2-z1)
    dist = sqrt(distsquared)
    return dist
  end

  # this function takes a point, a unit vector, and a distance, and adds the distance to the point in the direction of the unit vector (3d space)
  # it returns a point as a list of coordinates
  def add_vectordistance_to_point(xi, yi, zi, uvx, uvy, uvz, delta):
    xf = xi + uvx * delta
    yf = yi + uvy * delta
    zf = zi + uvz * delta
    ret = [xf, yf, zf]
    return ret
  end

  # this function converts a heading (ccw radians from the positive x axis) into rxryrz to be put into a point p[]
  # this will point the gun in this heading with the bottom side of the gun facing up.
  # the values used in this program were calculated by doing rotation matrix math in the file on WI-CALVINB10 C. Documents. Theory for converting rotations into axis angle representations
  def convert_heading_to_axang(heading):
   axisxraw = -1 * sin(heading)
   axisyraw = cos(heading) + 1
   axiszraw = sin(heading)

   magnitude = sqrt(axisxraw*axisxraw + axisyraw*axisyraw + axiszraw*axiszraw)

   axisxunit = axisxraw / magnitude
   axisyunit = axisyraw / magnitude
   axiszunit = axiszraw / magnitude

   angle = acos( (cos(heading) - 1) / 2 )

   rxout = axisxunit * angle
   ryout = axisyunit * angle
   rzout = axiszunit * angle

   return [rxout, ryout, rzout]
  end

  # this function converts a heading (ccw radians from the positive x axis) into rxryrz to be put into a point p[]
  # this will point the gun in this heading with the preheat side of the gun tip facing up. Used for welding in a vertical path.
  # the values used in this program were calculated by doing rotation matrix math in the file on WI-CALVINB10 C. Documents. Theory for converting rotations into axis angle representations
  def convert_heading_to_axang_preheatup(heading):
   axisxraw = -sin(heading) + 1
   axisyraw = cos(heading)
   axiszraw = cos(heading)

   magnitude = sqrt(axisxraw*axisxraw + axisyraw*axisyraw + axiszraw*axiszraw)

   axisxunit = axisxraw / magnitude
   axisyunit = axisyraw / magnitude
   axiszunit = axiszraw / magnitude

   angle = acos( (-sin(heading) - 1) / 2 )

   rxout = axisxunit * angle
   ryout = axisyunit * angle
   rzout = axiszunit * angle

   return [rxout, ryout, rzout]
  end

  # this function converts a heading (ccw radians from the positive x axis) into rxryrz to be put into a point p[]
  # this will point the gun in this heading with the preheat side of the gun tip facing down. Used for welding in a vertical path downwards.
  # the values used in this program were calculated by doing rotation matrix math in the file on WI-CALVINB10 C. Documents. Theory for converting rotations into axis angle representations
  def convert_heading_to_axang_preheatdown(heading):
   axisxraw = -sin(heading) - 1
   axisyraw = cos(heading)
   axiszraw = -cos(heading)

   magnitude = sqrt(axisxraw*axisxraw + axisyraw*axisyraw + axiszraw*axiszraw)

   axisxunit = axisxraw / magnitude
   axisyunit = axisyraw / magnitude
   axiszunit = axiszraw / magnitude

   angle = acos( (sin(heading) - 1) / 2 )

   rxout = axisxunit * angle
   ryout = axisyunit * angle
   rzout = axiszunit * angle

   return [rxout, ryout, rzout]
  end

  # this function converts a heading (ccw radians from the positive x axis) into rxryrz to be put into a point p[]
  # this will point the gun in this heading with the preheat side of the gun tip facing right. Used for welding counterclockwise around the box.
  # the values used in this program were calculated by doing rotation matrix math in the file on WI-CALVINB10 C. Documents. Theory for converting rotations into axis angle representations
  def convert_heading_to_axang_ccw(heading):
   axisxraw = -sin(heading)
   axisyraw = cos(heading) - 1
   axiszraw = -sin(heading)

   magnitude = sqrt(axisxraw*axisxraw + axisyraw*axisyraw + axiszraw*axiszraw)

   axisxunit = axisxraw / magnitude
   axisyunit = axisyraw / magnitude
   axiszunit = axiszraw / magnitude

   angle = acos( (-cos(heading) - 1) / 2 )

   rxout = axisxunit * angle
   ryout = axisyunit * angle
   rzout = axiszunit * angle

   return [rxout, ryout, rzout]
  end

  # this function is for getting the points along the path of the corner homing 45
  # point0 is the point where they touched
  def get_corner_homing_45_pathpoints(point0):
    p0x = point0[0]
    p0y = point0[1]
    p0z = point0[2]
    p0rx = point0[3]
    p0ry = point0[4]
    p0rz = point0[5]

    #constants
    #distances of how far away from point the touchpoints are
    d0 = 0.15 # how far from the box to retreat and approach
    d1 = 0.05
    d2 = 0.2
    sqrt2 = 0.707106781

    ph1 = p[p0x + d0, p0y, p0z + .05, p0rx, p0ry, p0rz] #approach point for turn

    ph2 = p[p0x+d0-d0*sqrt2-sqrt2*d1, p0y+d0*sqrt2+sqrt2*d1, p0z+.05, .445, -1.562, .483]
    ph3 = p[p0x+d0-d0*sqrt2-sqrt2*d2, p0y+d0*sqrt2+sqrt2*d2, p0z+.05, .445, -1.562, .483]
    ph4 = p[p0x+d0-d0*sqrt2-sqrt2*d1, p0y-d0*sqrt2-sqrt2*d1, p0z+.05, 1.699, 3.576, 1.841]
    ph5 = p[p0x+d0-d0*sqrt2-sqrt2*d2, p0y-d0*sqrt2-sqrt2*d2, p0z+.05, 1.699, 3.576, 1.841]

    # go back to ph1
    ph6 = p[p0x + .05, p0y, p0z -.05, 0, 0, 0] # approach point for under turn
    # moveL from ph1 to ph6
    ph7 = p[p0x-.05, p0y, p0z-.05, 0, 0, 0]
    ret = struct(ph1=ph1, ph2=ph2, ph3=ph3, ph4=ph4, ph5=ph5, ph6=ph6, ph7=ph7)
    return ret
  end
  $ 16 "pathturn≔main_calculate_right(p11,p12,p21,p22,p3)"
  global pathturn=main_calculate_right(p11,p12,p21,p22,p3)
  $ 18 "Call move_path_3right"
  move_path_3right()
  $ 19 "Home"
  movej([-3.4579734502641006, -2.05691362454537, 2.326567589830591, -0.22707360390354125, -0.19934432301767302, -0.10534790278823536], a=1.3962634015954636, v=1.0471975511965976)
end
